// TIA Portal V19 export
FUNCTION_BLOCK "A0302_Manager_FB"   // FB51, LAD
// stored: MemoryReserve 100, SetENOAutomatically false
   VAR_INPUT
      AreaInterface : "AreaInterface";
      DataIn : Struct
         SemiAut_Pb : Bool;
      END_STRUCT;
      CIn : Struct
         P5 : Struct
            Sollevatori { ExternalAccessible := 'False'; ExternalVisible := 'False'; ExternalWritable := 'False'} : "ValveMachine_COut";
            Spintore_Lat : Struct
               Spin_Lat1 : Struct
                  Standstill : Bool;
                  Rest_CheckNext : Bool;
                  Work_CheckNext : Bool;
                  Rest : Bool;
                  Work : Bool;
               END_STRUCT;
               Spin_Lat2 : Struct
                  Standstill : Bool;
                  Rest_CheckNext : Bool;
                  Work_CheckNext : Bool;
                  Rest : Bool;
                  Work : Bool;
               END_STRUCT;
            END_STRUCT;
            SpintoreLong { ExternalAccessible := 'False'; ExternalVisible := 'False'; ExternalWritable := 'False'} : Struct   // Spintore Longitudinale
               Ax : "Positioning_EPOS_Machine_COut";
               Ax_Sts : Struct
                  PosAttesa_Reached : Bool;
                  PosFineSpinta_Reached : Bool;
               END_STRUCT;
               Spintore : "ValveMachine_COut";
               Vrt : "ValveMachine_COut";
               Orz : "ValveMachine_COut";
               Sens : Struct
                  FTC_FuoriIngombro : Bool;
               END_STRUCT;
            END_STRUCT;
         END_STRUCT;
         Bordatrice : Struct
            Ax : "Positioning_EPOS_Machine_COut";
            Sts : Struct
               PosTargetEnable : Bool;
               PosTarget_Reached : Bool;
               In_W_Pos : Bool;
               AtRest : Bool;
            END_STRUCT;
            Sens : Struct
               FTC_Ingresso : Bool;   // 1833SQ1 - I46.0 (Predisposta - usiamo la 1614BF1)
               FTC_Uscita : Bool;
            END_STRUCT;
         END_STRUCT;
         Rulliera { ExternalAccessible := 'False'; ExternalVisible := 'False'; ExternalWritable := 'False'} : Struct
            Ax_1 : "SpeedMachine_COut";
            Ax_2 : "SpeedMachine_COut";
            Centraggio : "ValveMachine_COut";   // Chiusura Centratori
            Sollevamento : "ValveMachine_COut";   // Solleva centratori
            Coda : Struct
               Sens : Struct
                  FTC_Rall : Bool;   // Sensori presenza materiale banco rallentamento ingresso
                  FTC_Prox_Ing : Bool;   // Sensori presenza materiale banco limite ingresso
               END_STRUCT;
            END_STRUCT;
            Centro : Struct
               Sens : Struct
                  FTC_Centrale : Bool;
               END_STRUCT;
            END_STRUCT;
         END_STRUCT;
         CarroPareggCoda { ExternalAccessible := 'False'; ExternalVisible := 'False'; ExternalWritable := 'False'} : Struct
            Ax_InWPos : Bool;
            Ax : "Positioning_DOL_Machine_COut";
            Bloccaggio : "ValveMachine_COut";
            BattutaVerticale : "ValveMachine_COut";
            PareggiatoreLong : "ValveMachine_COut";
            Sens : Struct
               FTC_Ingombro_Ing : Bool;   // FTC fuori ingombro lato ingresso al carro pareggiatore di coda
               FTC_Ingombro_Out : Bool;   // FTC fuori ingombro lato uscita al carro pareggiatore di coda
               PresenzaMat : Bool;   // FC presenza materiale agganciato
               PosPareggLong : Struct
                  Value : LReal;
                  CheckMeasure : Bool;
                  Standstill : Bool;
               END_STRUCT;
            END_STRUCT;
         END_STRUCT;
         CarroPareggTesta { ExternalAccessible := 'False'; ExternalVisible := 'False'; ExternalWritable := 'False'} : Struct
            Ax_InWPos : Bool;
            Ax : "Positioning_DOL_Machine_COut";
            Bloccaggio : "ValveMachine_COut";
            Centraggio : "ValveMachine_COut";
            Sollevatore : "ValveMachine_COut";
            Sens : Struct
               FTC_Ingombro_Ing : Bool;   // FTC fuori ingombro lato ingresso al carro pareggiatore di testa - Rallentamento rulliera
               FTC_Prox_Ls : Bool;   // FTC sensore presenza materiale banco limite ingresso
               PresenzaMat : Bool;   // FC presenza materiale agganciato
            END_STRUCT;
         END_STRUCT;
         Manipolatori : Struct
            Testa : Struct
               Ax : "Positioning_EPOS_Machine_COut";
               Sollevatore : "ValveMachine_COut";
               Magnete : "ValveMachine_COut";
            END_STRUCT;
            Coda : Struct
               Ax : "Positioning_EPOS_Machine_COut";
               Sollevatore : "ValveMachine_COut";
               Magnete : "ValveMachine_COut";
            END_STRUCT;
            InPos_Prelievo : Bool;
            InPos_BancoScarto : Bool;
            InPos_BancoA0303 : Bool;
         END_STRUCT;
         Spalle : Struct
            Coda : Struct
               Ax : "Positioning_DOL_Machine_COut";
            END_STRUCT;
            Testa : Struct
               Ax : "Positioning_DOL_Machine_COut";
            END_STRUCT;
         END_STRUCT;
         Banco_A0303 : Struct
            ReadyToRecive : Bool;   // Consenso da Stazione A0303 a ricevere il pezzo buono misurato
         END_STRUCT;
         ProdManager : "Prod_Beam_Ctrl";
      END_STRUCT;
   END_VAR
   VAR_OUTPUT
      MachineInterface : "MachineInterface";
      COut : Struct
         HU : Struct
            EnableStopDoorOpeningReq : Bool;
            EnableStopInPhase : Bool;
            EnableStopProgrammed : Bool;
            Control_ON : Bool;
            Rest : Bool;
            Work : Bool;
         END_STRUCT;
         SpintoreLong : Struct
            EnableStopDoorOpeningReq : Bool;
            EnableStopInPhase : Bool;
            EnableStopProgrammed : Bool;
            Control_ON : Bool;
            REST_Req : Bool;
            WORK_Req : Bool;
            Rest : Bool;
            Work : Bool;
         END_STRUCT;
         Bordatrice : Struct
            Ax : "Positioning_EPOS_Machine_Manager";
            Sts : Struct
               PosTarget_Reached : Bool;
               AtRest : Bool;
            END_STRUCT;
            DataOut : "Positioning_EPOS_Machine_DataOut";
            Rest_Req : Bool;
            Work_Req : Bool;
         END_STRUCT;
         Rulliera : Struct
            Ax_1 : "SpeedMachine_CIn_Manager";
            Ax_2 : "SpeedMachine_CIn_Manager";
            Centratori : Struct   // Chiusura Centratori
               Sollevamento : "ValveMachine_Manager";
               Centraggio : "ValveMachine_Manager";
            END_STRUCT;
            Ax_1_Frw_Req : Bool;
            Ax_1_Brw_Req : Bool;
            Ax_2_Frw_Req : Bool;
            Ax_2_Brw_Req : Bool;
         END_STRUCT;
         CarroPareggCoda : Struct
            EnableStopDoorOpeningReq : Bool;
            EnableStopInPhase : Bool;
            EnableStopProgrammed : Bool;
            Control_ON : Bool;
            MoveToPos : Bool;
            Pos : LReal;
            Speed : LReal;
            Bloccaggio : Struct
               Rest : Bool;
               Work : Bool;
            END_STRUCT;
            BattutaVrt : Struct
               Rest : Bool;
               Work : Bool;
            END_STRUCT;
            PareggLong : Struct
               Rest : Bool;
               Work : Bool;
            END_STRUCT;
         END_STRUCT;
         CarroPareggTesta : Struct
            EnableStopDoorOpeningReq : Bool;
            EnableStopInPhase : Bool;
            EnableStopProgrammed : Bool;
            Control_ON : Bool;
            MoveToPos : Bool;
            Pos : LReal;
            Speed : LReal;
            Bloccaggio : "OP_PB";
            Sollevamento : "OP_PB";
            Centraggio : "OP_PB";
         END_STRUCT;
         Manipolatori : Struct
            Ax : Struct
               EnableStopDoorOpeningReq : Bool;
               EnableStopInPhase : Bool;
               EnableStopProgrammed : Bool;
               Control_ON : Bool;
               MoveToPos : Bool;
               Pos : LReal;
               Vel : LReal;
               Acc : LReal;
               Dec : LReal;
            END_STRUCT;
            Sollevatori : "OP_PB";
            Magneti : "OP_PB";
         END_STRUCT;
      END_STRUCT;
   END_VAR
   VAR_IN_OUT
      Par : Struct
         CarroPareggCoda : Struct
            Delay_StartMove : Time;
            Preset : LReal;
         END_STRUCT;
         CarroPareggTesta : Struct
            Delay_StartMove : Time;
            Preset : LReal;
         END_STRUCT;
         Cremaliera : Struct
            Modulo : LReal;
            Passo : LReal;
         END_STRUCT;
      END_STRUCT;
   END_VAR
   VAR
      Alarm : Struct
         Qlty_Unknow : Bool;   // Allarme pezzo sconosciuto
         ToCheckList_Full : Bool;
         WrongReadPz_ManipBasso : Bool;
         Pz_NonPareggiabile : Bool;
         STOP_FineTurno : Bool;
         STOP_End_Of_Proroduction : Bool;
         STOP_ControlloQualita : Bool;
      END_STRUCT;
      Warning : Struct
         CheckBancoAccumulo : Bool;
      END_STRUCT;
      Sts : Struct
         SemiAut : Struct
            ON : Bool;
            Request : Bool;
            MaterialFrw : Bool;
         END_STRUCT;
         CarroPareggTesta : Struct
            InCyclePos : Bool;
         END_STRUCT;
         CarroPareggCoda : Struct
            InCyclePos : Bool;
         END_STRUCT;
         Attrezzamento : Struct
            Ready : Bool;
            FindNewID : Bool;
            RequestNewPosition : Bool;
            OLD_OID : DInt;
         END_STRUCT;
         BTrk : Struct
            A0302Exit_Actual_O_ID : DInt;
            BLen_Paregg : Real;
            Last_Misure1Paregg : Real;
            Last_Misure2Paregg : Real;
            A0302Entry_Absence : Bool;
            A0302Exit_Absence : Bool;
            ZoneA0302Entry_Empty : Bool;
            ZoneA0302Exit_Empty : Bool;
            A0302_CheckBancoAccumulo : Bool;
            Waiting_A0302_Recive : Bool;
         END_STRUCT;
         AlarmsPresence : Bool;
         WarningsPresence : Bool;
         IsStandstill : Bool;
      END_STRUCT;
      Ctrl : Struct
         Stop : Bool;
         TRK : Struct
            BTrk : Struct
               "P5.1_To_LongPosAttesa" : Bool;
               "P5.2_LongPosAttesa_TO_Spintore" : Bool;
               "P5.2_Spintore_TO_ExitA031" : Bool;
               "P5.2_ExitA031_To_IngBord" : Bool;
               "P5.2_Ax_MoveToPosAttesa" : Bool;
               "P5.2_Ax_PreparingPosAttesa" : Bool;
               "P5.2_Ax_MoveToPosSpinta" : Bool;
               SpinBord_In_To_Bord_In : Bool;
               Bordatrice_In_To_Out : Bool;   // il pezzo ha raggiunto il sensore di uscita della bordatrice (xxxSQx) (salvataggio posizione asse bordatrice)
               Bordatrice_Out_To_PareggCodaUp : Bool;   // Il pezzo è in uscita della bordatrice e la posizione target non è limitata perchè il pareggiamento di coda è alto
               Bordatrice_Out_To_PareggCodaDown : Bool;   // Il pezzo è in uscita della bordatrice ma la posizione target è limitata per non collidere con il pareggiamento di coda basso
               Rulliera_Start_Brw : Bool;
               Rulliera_Ax_1_Start_Frw : Bool;
               Rulliera_Ax_2_Start_Frw : Bool;
               RulliereVode : Bool;
               PCodaDown_TO_Rulli_PCodaDown : Bool;   // Pezzo su rulliera (1) + pareggiatore coda basso quindi quando incontra sensore (1,2) deve rallentare
               PCodaDown_TO_RALL_Rulli_PCodaDown : Bool;   // Pezzo su rulliera (1) + pareggiatore coda basso e ha incontrato sensore (1,2) di rallentamento
               PCodaDown_TO_STOP_PCodaDown : Bool;   // Pezzo su rulliera (1) + pareggiatore coda basso e ha incontrato sensore (3) di stop
               STOP_PCodaDown_TO_PCoda_Up : Bool;   // Pezzo su rulliera (1) + pareggiatore coda alto quindi può muoversi liberamente
               "PareggCodaUp_To_Rull-PrimaPareggCodaAltro" : Bool;
               PCoda_Up_TO_PCoda_UP_S3 : Bool;   // Pezzo su rulliera (1) + pareggiatore coda alto ed ha incontrato il sensore 3 (in ingresso al pareg.)
               PCoda_UP_S3_TO_PCoda_UP_S4 : Bool;   // Pezzo su rulliera (1) + pareggiatore coda alto ed ha incontrato il sensore 4 (in uscita al pareg.)
               PCoda_UP_S4_TO_PCoda_DownCnd : Bool;   // Pezzo su rulliera (1/2) + pareggiatore coda che è alto ed ha liberato il sensore 4-> Pareg. può andare basso (posizione di lavoro)
               PCoda_Beam_TO_PTesta : Bool;   // Pezzo su rulliera (1/2) tra il pareggiatore di testa e quello di coda
               Beam_TO_Stop_PTesta : Bool;   // Pezzo su rulliera (1/2) + ha incontrato il sensore 5 su pareggiatore di testa
               "Stop_PTesta_TO_Rull-Centratori" : Bool;   // Pezzo su rulliera (1/2) tra i pareggiatori + centratori a lavoro
               "Rull-Centratori_TO_Cnd_PareggCoda" : Bool;   // Pezzo su rulliera (1/2) tra i pareggiatori (quello di coda è basso) + centratori a lavoro
               Cnd_PareggCoda_TO_Pareggiato : Bool;   // Pezzo su rulliera (1/2) tra i pareggiatori e paregiatura di coda eseguito lavoro cilindro idraulico (ora si sa la misura del pezzo, si può mettere utenze in attesa del prossimo pezzo)
               Check_Tolleranza_BLen_Qlty : Bool;
               Pareggiato_TO_PresaBasso : Bool;   // Pezzo su magneti del manipolatore basso in posizione di presa.
               PresaBasso_TO_PresaAlto : Bool;   // Pezzo su magneti del manipolatore alto in posizione di presa.
               PresaAlto_To_CheckOut_BadQlty : Bool;   // Pezzo su magneti del manipolatore alto in posizione di uscita perchè non conforme
               CheckOut_BadQlty_UP_MoveToPos : Bool;   // Ho il pezzo in presa alta > vado in posizione uscita banco scarto
               PresaAlto_To_CheckOut_GoodQlty : Bool;   // Pezzo su magneti del manipolatore alto in posizione per deposito su A0303
               CheckOut_GoodQlty_UP_MoveToPos : Bool;   // Ho il pezzo in presa alta > vado in posizione uscita banco A0303
               CheckOut_BadQlty_UP_To_DOWN : Bool;   // Pezzo su magneti del manipolatore basso in posizione di uscita perchè non conforme
               CheckOut_BadQlty_DOWN_To_Sgancia : Bool;
               CheckOut_GoodQlty_UP_To_DOWN : Bool;   // Pezzo su magneti del manipolatore basso in posizione per deposito su A0303
               CheckOut_GoodQlty_DOWN_To_Sgancia : Bool;
               Manipolatori_Return_ToPrelievo : Bool;   // Ritorno degli assi manipolatore a zero e / o a prelievo
            END_STRUCT;
            BTrk_ToCheck : Struct
               ClearList : Bool;
               QtyClear_RetVal : Bool;
               Prelievo_RecondGood : Bool;   // Attivo durante la fase di posizionamento manuale del Beam fino a quando il manipolatore lo prende
               RecG_InPos_Centraggio : Bool;   // Beam ricondizionato posizionato su rulliera da centrare
               RegG_InPos_ReadyPickUp : Bool;
            END_STRUCT;
         END_STRUCT;
         SpintoreLong : Struct
            Rest : Bool;
            Work : Bool;
            MoveAttesaDisable : Bool;
         END_STRUCT;
         Bordatrice : Struct
            Run : Bool;
         END_STRUCT;
         Rulliera : Struct
            Ax_1_Vel_Bord : Bool;
            Ax_2_Vel_Bord : Bool;
            Ax_1_Lenta_CarroCoda : Bool;
            Ax_1_2_Vel_CarroTesta : Bool;
            Ax_1_2_Vel_ZeroTesta : Bool;
            Ax_1_2_Vel_Appoggio : Bool;
            Ax_1_2_End_VelZero : Bool;
            Ax_2_MemoRall : Bool;
            SP_TimeMemoRall : Time;
            TON_RitardoRallenta : IEC_TIMER;
            Centraggio : Struct
               Rest : Bool;
               Work : Bool;
            END_STRUCT;
            Sollevamento : Struct
               Rest : Bool;
               Work : Bool;
            END_STRUCT;
         END_STRUCT;
         CarroPareggCoda : Struct
            Ax : Struct
               MoveToPos : Bool;
               Pos : LReal;
            END_STRUCT;
            Bloccaggio : Struct
               Rest : Bool;
               Work : Bool;
            END_STRUCT;
            BattutaVerticale : Struct
               Rest : Bool;
               Work : Bool;
            END_STRUCT;
            PareggiatoreLong : Struct
               Rest : Bool;
               Work : Bool;
            END_STRUCT;
            MisuraPzPareggiato : Bool;
         END_STRUCT;
         CarroPareggTesta : Struct
            Ax : Struct
               MoveToPos : Bool;
               Pos : LReal;
            END_STRUCT;
            Bloccaggio : Struct
               Rest : Bool;
               Work : Bool;
            END_STRUCT;
            Sollevatore : Struct
               Rest : Bool;
               Work : Bool;
            END_STRUCT;
            Centraggio : Struct
               Rest : Bool;
               Work : Bool;
            END_STRUCT;
         END_STRUCT;
         Manipolatori : Struct
            Ax : Struct
               MoveToPos : Bool;
               Pos : LReal;
            END_STRUCT;
            Sollevatori : Struct
               Rest : Bool;
               Work : Bool;
            END_STRUCT;
            Magneti : Struct
               Rest : Bool;
               Work : Bool;
            END_STRUCT;
         END_STRUCT;
      END_STRUCT;
      HMI : Struct
         PlsClear_ListToCheck : Bool;
      END_STRUCT;
      BTrk_A0302_Exit_Item : Struct
         BLean : Real;
         W_A : Real;
         Tol_Max : Real;
         Tol_Min : Real;
         Good { ExternalAccessible := 'False'; ExternalVisible := 'False'; ExternalWritable := 'False'} : Bool;
         ToCheckLen { ExternalAccessible := 'False'; ExternalVisible := 'False'; ExternalWritable := 'False'} : Bool;
      END_STRUCT;
      BTrk_ListToCheck : Struct
         Recond : Struct
            Found : Bool;
            Nr_B : Int;
         END_STRUCT;
      END_STRUCT;
      OffsetCarri : Struct
         DaSpallaTesta : LReal;
         DaSpallaCoda : LReal;
      END_STRUCT;
      CarroTesta : Struct
         RimanenzaPos : LReal;
         PassoReq : LReal;
         PosBattutePz : LReal;
         SemiBeamLen : LReal;
         NrPassiReq : LReal;
      END_STRUCT;
      CarroCoda : Struct
         RimanenzaPos : LReal;
         PassoReq : LReal;
         PosBattutePz : LReal;
         SemiBeamLen : LReal;
         NrPassiReq : LReal;
      END_STRUCT;
      TON_AlarmWrongReadPz_Manip : IEC_TIMER;
      TON_Alarm_FTC_CarroCodaOut { S7_SetPoint := 'True'} : IEC_TIMER;
      TON_Stop { S7_SetPoint := 'True'} : IEC_TIMER;
   END_VAR
   VAR_TEMP
      AUX : Struct
         SemiAut_Pb : Bool;
      END_STRUCT;
      i : Int;
      BTrk_A0302_EXIT_GetData : Struct   // Appoggio struttura per lettura dati dal Mes
         indx : Int;   // Se trovato tra i TODO / ENDING / OUT questo è l'indice dove sono stati prelevati i dati
         Sts : Int;   // 0 = Non Trovato; 0 = ACT; 1 = TODO; 2=ENDING; 3 = OUT
         Item : "Prod_Item_small";
      END_STRUCT;
      DisableA0302 : Bool;
      PieceToCheck_Presence : Bool;
      CarroTestaCentraggio_Disable : Bool;
   END_VAR
   VAR CONSTANT
      OffsetGioco : Real := 2.0;   // Offset gioco carri durante lettura Pareggiamento pezzo
   END_VAR
   VAR_TEMP   // added for the SCL form of the ladder/FBD networks
      _w1 : Bool;
      _w2 : Bool;
      _w3 : Bool;
      _w4 : Bool;
      _w5 : Bool;
      _w6 : Bool;
      _w7 : Bool;
      _w8 : Bool;
      _w9 : Bool;
      _w10 : Bool;
      _w11 : Bool;
      _w12 : Bool;
      _w13 : Bool;
      _w14 : Bool;
      _w15 : Bool;
      _w16 : Bool;
      _w17 : Bool;
      _w18 : Bool;
      _w19 : Bool;
      _w20 : Bool;
   END_VAR
BEGIN

REGION Network 1 (SCL): = Area - Rst =
   IF #AreaInterface.RstAlarms THEN
       #Alarm.Qlty_Unknow := FALSE;
       #Alarm.ToCheckList_Full := FALSE;
       #Alarm.STOP_ControlloQualita := FALSE;
       #Alarm.STOP_FineTurno := FALSE;
       #Alarm.STOP_End_Of_Proroduction := FALSE;
   END_IF;

   IF #AreaInterface.RstAlarms AND #CIn.CarroPareggCoda.Sens.PresenzaMat AND #CIn.CarroPareggTesta.Sens.PresenzaMat
       AND #CIn.Manipolatori.Testa.Magnete.Work AND #CIn.Manipolatori.Coda.Magnete.Work THEN
       #Alarm.WrongReadPz_ManipBasso := FALSE;
   END_IF;

   IF #AreaInterface.RstAlarms AND NOT #CIn.CarroPareggCoda.Sens.FTC_Ingombro_Out THEN
       #Alarm.Pz_NonPareggiabile := FALSE;
   END_IF;
END_REGION

REGION Network 2: ******** CLEAR TRACKING ARRIVATO ********
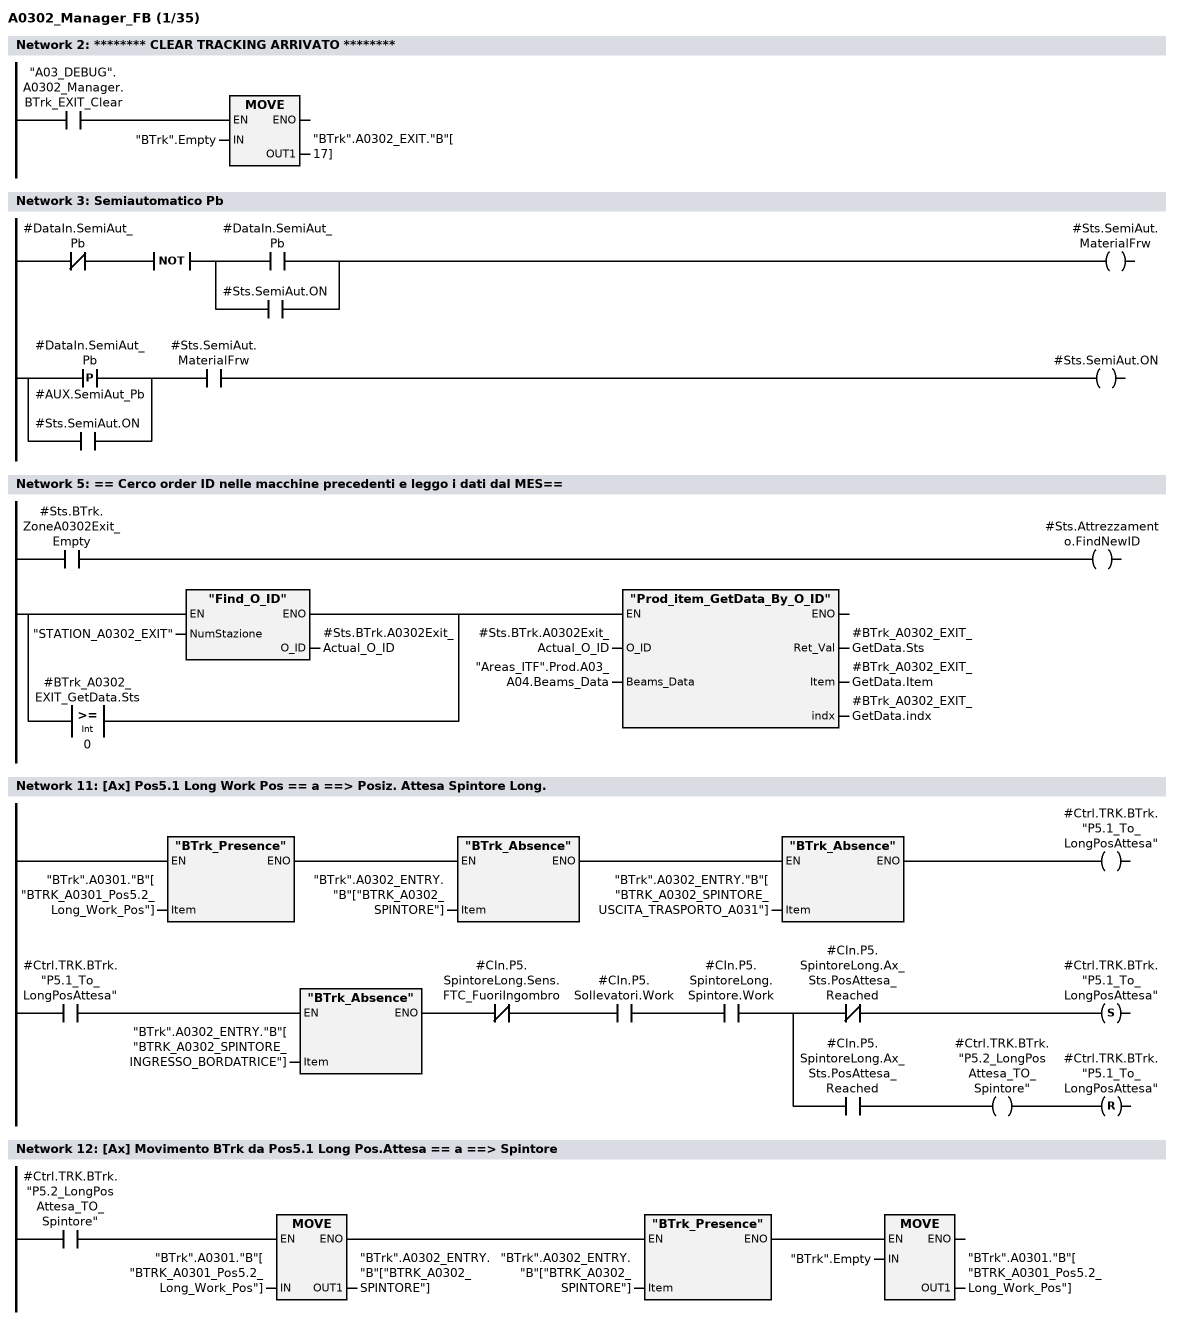
   RUNG wire#powerrail
      Contact( "A03_DEBUG".A0302_Manager.BTrk_EXIT_Clear )
      Move(in := "BTrk".Empty, out1 => "BTrk".A0302_EXIT."B"[17])
   END_RUNG
   // the same network as SCL:
   IF "A03_DEBUG".A0302_Manager.BTrk_EXIT_Clear THEN "BTrk".A0302_EXIT."B"[17] := "BTrk".Empty; END_IF;
END_REGION

REGION Network 3: Semiautomatico Pb
   RUNG wire#powerrail
      I_Contact( #DataIn.SemiAut_Pb )
      Not()
      wire#w1
      Contact( #DataIn.SemiAut_Pb )
      wire#w2
      Coil( #Sts.SemiAut.MaterialFrw )
   END_RUNG
   RUNG wire#w1
      Contact( #Sts.SemiAut.ON )
   END_RUNG wire#w2
   RUNG wire#powerrail
      P_Contact(operand := #DataIn.SemiAut_Pb, bit := #AUX.SemiAut_Pb)
      wire#w3
      Contact( #Sts.SemiAut.MaterialFrw )
      Coil( #Sts.SemiAut.ON )
   END_RUNG
   RUNG wire#powerrail
      Contact( #Sts.SemiAut.ON )
   END_RUNG wire#w3
   // the same network as SCL:
   #Sts.SemiAut.MaterialFrw := NOT (NOT #DataIn.SemiAut_Pb) AND (#DataIn.SemiAut_Pb OR #Sts.SemiAut.ON);
   #_w1 := #DataIn.SemiAut_Pb AND NOT #AUX.SemiAut_Pb;   // rising edge of #DataIn.SemiAut_Pb
   #AUX.SemiAut_Pb := #DataIn.SemiAut_Pb;
   #Sts.SemiAut.ON := (#_w1 OR #Sts.SemiAut.ON) AND #Sts.SemiAut.MaterialFrw;
END_REGION

REGION Network 5: == Cerco order ID nelle macchine precedenti e leggo i dati dal MES==
   RUNG wire#powerrail
      Contact( #Sts.BTrk.ZoneA0302Exit_Empty )
      Coil( #Sts.Attrezzamento.FindNewID )
   END_RUNG
   RUNG wire#powerrail
      "Find_O_ID"(NumStazione := "STATION_A0302_EXIT", O_ID => #Sts.BTrk.A0302Exit_Actual_O_ID)
      wire#w1
      "Prod_item_GetData_By_O_ID"(O_ID := #Sts.BTrk.A0302Exit_Actual_O_ID, Beams_Data := "Areas_ITF".Prod.A03_A04.Beams_Data, Ret_Val => #BTrk_A0302_EXIT_GetData.Sts, Item => #BTrk_A0302_EXIT_GetData.Item, indx => #BTrk_A0302_EXIT_GetData.indx)
   END_RUNG
   RUNG wire#powerrail
      { S7_Templates := "SrcType := Int" } GE_Contact(in1 := #BTrk_A0302_EXIT_GetData.Sts, in2 := 0)
   END_RUNG wire#w1
   // the same network as SCL:
   #Sts.Attrezzamento.FindNewID := #Sts.BTrk.ZoneA0302Exit_Empty;
   "Find_O_ID"(NumStazione := "STATION_A0302_EXIT", O_ID => #Sts.BTrk.A0302Exit_Actual_O_ID, ENO => #_w1);
   IF #_w1 OR (#BTrk_A0302_EXIT_GetData.Sts >= 0) THEN
       #BTrk_A0302_EXIT_GetData.Sts := "Prod_item_GetData_By_O_ID"(O_ID := #Sts.BTrk.A0302Exit_Actual_O_ID,
                               Beams_Data := "Areas_ITF".Prod.A03_A04.Beams_Data,
                               Item => #BTrk_A0302_EXIT_GetData.Item,
                               indx => #BTrk_A0302_EXIT_GetData.indx);
   END_IF;
END_REGION

REGION Network 6 (SCL): == Richiesta nuovo posizionamento carri Testa/Coda per cambio Traking ==

   //Se ho O_ID <> e non sono vuoto attivo avviso di attesa zona A0302 vuota
   IF (#Sts.BTrk.A0302Exit_Actual_O_ID <> #Sts.Attrezzamento.OLD_OID) OR (NOT #Sts.BTrk.ZoneA0302Exit_Empty OR NOT #Sts.BTrk.ZoneA0302Entry_Empty)THEN
       #Sts.BTrk.Waiting_A0302_Recive := TRUE;

   ELSIF (#Sts.BTrk.A0302Exit_Actual_O_ID = #Sts.Attrezzamento.OLD_OID) OR ( #Sts.BTrk.ZoneA0302Exit_Empty AND #Sts.BTrk.ZoneA0302Entry_Empty) THEN
       #Sts.BTrk.Waiting_A0302_Recive := FALSE;

   END_IF;

   //Se ho O_ID <> e sono vuoto aggiorno vecchio O_ID 
   IF (#Sts.BTrk.A0302Exit_Actual_O_ID <> #Sts.Attrezzamento.OLD_OID) AND #Sts.BTrk.ZoneA0302Exit_Empty AND #Sts.BTrk.ZoneA0302Entry_Empty THEN
       #Sts.Attrezzamento.OLD_OID := #Sts.BTrk.A0302Exit_Actual_O_ID;
   END_IF;
END_REGION

REGION Network 7 (SCL): == Compilo i dati del btrk in base all'order ID in arrivo ==

   IF #BTrk_A0302_EXIT_GetData.Sts >= 0 THEN

       "BTrk".A0302_EXIT.O_ID:="BTrk".A0302_ENTRY.O_ID := #Sts.Attrezzamento.OLD_OID;
       "BTrk".A0302_EXIT.Beam_Len := "BTrk".A0302_ENTRY.Beam_Len := #BTrk_A0302_EXIT_GetData.Item.Beams_Len;
       "BTrk".A0302_EXIT.Beam_W_A := "BTrk".A0302_ENTRY.Beam_W_A := #BTrk_A0302_EXIT_GetData.Item.Beams_W_A;
       "BTrk".A0302_EXIT.Beam_H_B := "BTrk".A0302_ENTRY.Beam_H_B := #BTrk_A0302_EXIT_GetData.Item.Beams_H_B;

   ELSE
           "BTrk".A0302_EXIT.O_ID := "BTrk".A0302_ENTRY.O_ID := "BTrk".A0301.O_ID := -1;
           "BTrk".A0302_EXIT.Beam_Len := "BTrk".A0302_ENTRY.Beam_Len := -1.0;
           "BTrk".A0302_EXIT.Beam_W_A := "BTrk".A0302_ENTRY.Beam_W_A := -1.0;
           "BTrk".A0302_EXIT.Beam_H_B := "BTrk".A0302_ENTRY.Beam_H_B := -1.0;
   END_IF;
END_REGION

REGION Network 8 (SCL): == Richiesta nuovo posizionamento x cambio Order ID ==

   #Sts.Attrezzamento.RequestNewPosition := ("BTrk".A0302_EXIT.O_ID <> -1)
   AND (#BTrk_A0302_EXIT_GetData.Sts >= 0)
   AND (#BTrk_A0302_EXIT_GetData.Item.Beam_Code = 1)
   AND #Sts.Attrezzamento.FindNewID
   AND NOT #Sts.Attrezzamento.Ready
   AND NOT #BTrk_ListToCheck.Recond.Found
   AND (NOT #CIn.CarroPareggCoda.Ax_InWPos OR NOT #CIn.CarroPareggTesta.Ax_InWPos);
END_REGION

REGION Network 10: <<<< SPINTORE LONGITUDINALE >>>>
END_REGION

REGION Network 11: [Ax] Pos5.1 Long Work Pos == a ==> Posiz. Attesa Spintore Long.
   RUNG wire#powerrail
      "BTrk_Presence"(Item := "BTrk".A0301."B"["BTRK_A0301_Pos5.2_Long_Work_Pos"])
      "BTrk_Absence"(Item := "BTrk".A0302_ENTRY."B"["BTRK_A0302_SPINTORE"])
      "BTrk_Absence"(Item := "BTrk".A0302_ENTRY."B"["BTRK_A0302_SPINTORE_USCITA_TRASPORTO_A031"])
      Coil( #Ctrl.TRK.BTrk."P5.1_To_LongPosAttesa" )
   END_RUNG
   RUNG wire#powerrail
      Contact( #Ctrl.TRK.BTrk."P5.1_To_LongPosAttesa" )
      "BTrk_Absence"(Item := "BTrk".A0302_ENTRY."B"["BTRK_A0302_SPINTORE_INGRESSO_BORDATRICE"])
      I_Contact( #CIn.P5.SpintoreLong.Sens.FTC_FuoriIngombro )
      Contact( #CIn.P5.Sollevatori.Work )
      Contact( #CIn.P5.SpintoreLong.Spintore.Work )
      wire#w1
      I_Contact( #CIn.P5.SpintoreLong.Ax_Sts.PosAttesa_Reached )
      S_Coil( #Ctrl.TRK.BTrk."P5.1_To_LongPosAttesa" )
   END_RUNG
   RUNG wire#w1
      Contact( #CIn.P5.SpintoreLong.Ax_Sts.PosAttesa_Reached )
      Coil( #Ctrl.TRK.BTrk."P5.2_LongPosAttesa_TO_Spintore" )
      R_Coil( #Ctrl.TRK.BTrk."P5.1_To_LongPosAttesa" )
   END_RUNG
   // the same network as SCL:
   "BTrk_Presence"(Item := "BTrk".A0301."B"["BTRK_A0301_Pos5.2_Long_Work_Pos"], ENO => #_w1);
   "BTrk_Absence"(EN := #_w1, Item := "BTrk".A0302_ENTRY."B"["BTRK_A0302_SPINTORE"], ENO => #_w2);
   "BTrk_Absence"(EN := #_w2,
                  Item := "BTrk".A0302_ENTRY."B"["BTRK_A0302_SPINTORE_USCITA_TRASPORTO_A031"],
                  ENO => #_w3);
   #Ctrl.TRK.BTrk."P5.1_To_LongPosAttesa" := #_w3;
   "BTrk_Absence"(EN := #Ctrl.TRK.BTrk."P5.1_To_LongPosAttesa",
                  Item := "BTrk".A0302_ENTRY."B"["BTRK_A0302_SPINTORE_INGRESSO_BORDATRICE"],
                  ENO => #_w4);
   #_w5 := #_w4 AND NOT #CIn.P5.SpintoreLong.Sens.FTC_FuoriIngombro AND #CIn.P5.Sollevatori.Work AND #CIn.P5.SpintoreLong.Spintore.Work;
   IF #_w5 AND NOT #CIn.P5.SpintoreLong.Ax_Sts.PosAttesa_Reached THEN
       #Ctrl.TRK.BTrk."P5.1_To_LongPosAttesa" := TRUE;
   END_IF;
   #Ctrl.TRK.BTrk."P5.2_LongPosAttesa_TO_Spintore" := #_w5 AND #CIn.P5.SpintoreLong.Ax_Sts.PosAttesa_Reached;
   IF #Ctrl.TRK.BTrk."P5.2_LongPosAttesa_TO_Spintore" THEN
       #Ctrl.TRK.BTrk."P5.1_To_LongPosAttesa" := FALSE;
   END_IF;
END_REGION

REGION Network 12: [Ax] Movimento BTrk da Pos5.1 Long Pos.Attesa == a ==> Spintore
   RUNG wire#powerrail
      Contact( #Ctrl.TRK.BTrk."P5.2_LongPosAttesa_TO_Spintore" )
      Move(in := "BTrk".A0301."B"["BTRK_A0301_Pos5.2_Long_Work_Pos"], out1 => "BTrk".A0302_ENTRY."B"["BTRK_A0302_SPINTORE"])
      "BTrk_Presence"(Item := "BTrk".A0302_ENTRY."B"["BTRK_A0302_SPINTORE"])
      Move(in := "BTrk".Empty, out1 => "BTrk".A0301."B"["BTRK_A0301_Pos5.2_Long_Work_Pos"])
   END_RUNG
   // the same network as SCL:
   IF #Ctrl.TRK.BTrk."P5.2_LongPosAttesa_TO_Spintore" THEN
       "BTrk".A0302_ENTRY."B"["BTRK_A0302_SPINTORE"] := "BTrk".A0301."B"["BTRK_A0301_Pos5.2_Long_Work_Pos"];
   END_IF;
   "BTrk_Presence"(EN := #Ctrl.TRK.BTrk."P5.2_LongPosAttesa_TO_Spintore",
                   Item := "BTrk".A0302_ENTRY."B"["BTRK_A0302_SPINTORE"],
                   ENO => #_w1);
   IF #_w1 THEN "BTrk".A0301."B"["BTRK_A0301_Pos5.2_Long_Work_Pos"] := "BTrk".Empty; END_IF;
END_REGION

REGION Network 13: [Ax] Movimento BTrk da A3202 Spintore ==a==> Uscita Trasporto A031
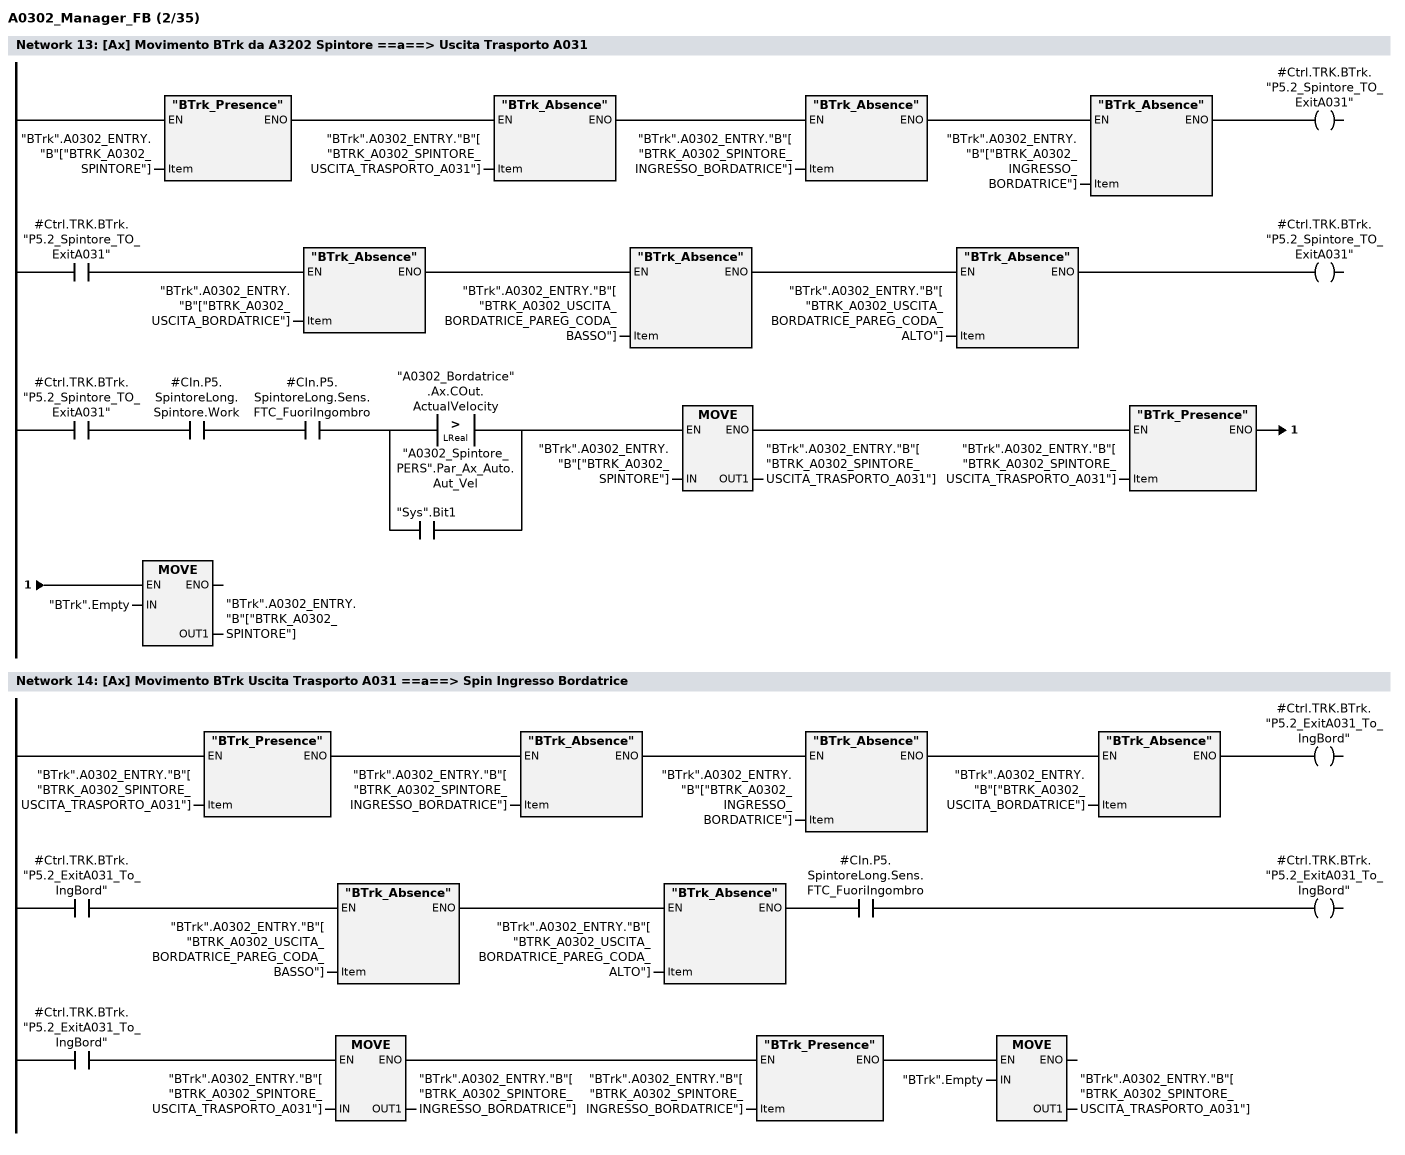
   RUNG wire#powerrail
      "BTrk_Presence"(Item := "BTrk".A0302_ENTRY."B"["BTRK_A0302_SPINTORE"])
      "BTrk_Absence"(Item := "BTrk".A0302_ENTRY."B"["BTRK_A0302_SPINTORE_USCITA_TRASPORTO_A031"])
      "BTrk_Absence"(Item := "BTrk".A0302_ENTRY."B"["BTRK_A0302_SPINTORE_INGRESSO_BORDATRICE"])
      "BTrk_Absence"(Item := "BTrk".A0302_ENTRY."B"["BTRK_A0302_INGRESSO_BORDATRICE"])
      Coil( #Ctrl.TRK.BTrk."P5.2_Spintore_TO_ExitA031" )
   END_RUNG
   RUNG wire#powerrail
      Contact( #Ctrl.TRK.BTrk."P5.2_Spintore_TO_ExitA031" )
      "BTrk_Absence"(Item := "BTrk".A0302_ENTRY."B"["BTRK_A0302_USCITA_BORDATRICE"])
      "BTrk_Absence"(Item := "BTrk".A0302_ENTRY."B"["BTRK_A0302_USCITA_BORDATRICE_PAREG_CODA_BASSO"])
      "BTrk_Absence"(Item := "BTrk".A0302_ENTRY."B"["BTRK_A0302_USCITA_BORDATRICE_PAREG_CODA_ALTO"])
      Coil( #Ctrl.TRK.BTrk."P5.2_Spintore_TO_ExitA031" )
   END_RUNG
   RUNG wire#powerrail
      Contact( #Ctrl.TRK.BTrk."P5.2_Spintore_TO_ExitA031" )
      Contact( #CIn.P5.SpintoreLong.Spintore.Work )
      Contact( #CIn.P5.SpintoreLong.Sens.FTC_FuoriIngombro )
      wire#w1
      { S7_Templates := "SrcType := LReal" } GT_Contact(in1 := "A0302_Bordatrice".Ax.COut.ActualVelocity, in2 := "A0302_Spintore_PERS".Par_Ax_Auto.Aut_Vel)
      wire#w2
      Move(in := "BTrk".A0302_ENTRY."B"["BTRK_A0302_SPINTORE"], out1 => "BTrk".A0302_ENTRY."B"["BTRK_A0302_SPINTORE_USCITA_TRASPORTO_A031"])
      "BTrk_Presence"(Item := "BTrk".A0302_ENTRY."B"["BTRK_A0302_SPINTORE_USCITA_TRASPORTO_A031"])
      Move(in := "BTrk".Empty, out1 => "BTrk".A0302_ENTRY."B"["BTRK_A0302_SPINTORE"])
   END_RUNG
   RUNG wire#w1
      Contact( "Sys".Bit1 )
   END_RUNG wire#w2
   // the same network as SCL:
   "BTrk_Presence"(Item := "BTrk".A0302_ENTRY."B"["BTRK_A0302_SPINTORE"], ENO => #_w1);
   "BTrk_Absence"(EN := #_w1,
                  Item := "BTrk".A0302_ENTRY."B"["BTRK_A0302_SPINTORE_USCITA_TRASPORTO_A031"],
                  ENO => #_w2);
   "BTrk_Absence"(EN := #_w2,
                  Item := "BTrk".A0302_ENTRY."B"["BTRK_A0302_SPINTORE_INGRESSO_BORDATRICE"],
                  ENO => #_w3);
   "BTrk_Absence"(EN := #_w3, Item := "BTrk".A0302_ENTRY."B"["BTRK_A0302_INGRESSO_BORDATRICE"], ENO => #_w4);
   #Ctrl.TRK.BTrk."P5.2_Spintore_TO_ExitA031" := #_w4;
   "BTrk_Absence"(EN := #Ctrl.TRK.BTrk."P5.2_Spintore_TO_ExitA031",
                  Item := "BTrk".A0302_ENTRY."B"["BTRK_A0302_USCITA_BORDATRICE"],
                  ENO => #_w5);
   "BTrk_Absence"(EN := #_w5,
                  Item := "BTrk".A0302_ENTRY."B"["BTRK_A0302_USCITA_BORDATRICE_PAREG_CODA_BASSO"],
                  ENO => #_w6);
   "BTrk_Absence"(EN := #_w6,
                  Item := "BTrk".A0302_ENTRY."B"["BTRK_A0302_USCITA_BORDATRICE_PAREG_CODA_ALTO"],
                  ENO => #_w7);
   #Ctrl.TRK.BTrk."P5.2_Spintore_TO_ExitA031" := #_w7;
   IF #Ctrl.TRK.BTrk."P5.2_Spintore_TO_ExitA031" AND #CIn.P5.SpintoreLong.Spintore.Work AND #CIn.P5.SpintoreLong.Sens.FTC_FuoriIngombro AND (("A0302_Bordatrice".Ax.COut.ActualVelocity > "A0302_Spintore_PERS".Par_Ax_Auto.Aut_Vel) OR "Sys".Bit1) THEN
       "BTrk".A0302_ENTRY."B"["BTRK_A0302_SPINTORE_USCITA_TRASPORTO_A031"] := "BTrk".A0302_ENTRY."B"["BTRK_A0302_SPINTORE"];
   END_IF;
   "BTrk_Presence"(EN := #Ctrl.TRK.BTrk."P5.2_Spintore_TO_ExitA031" AND #CIn.P5.SpintoreLong.Spintore.Work AND #CIn.P5.SpintoreLong.Sens.FTC_FuoriIngombro AND (("A0302_Bordatrice".Ax.COut.ActualVelocity > "A0302_Spintore_PERS".Par_Ax_Auto.Aut_Vel) OR "Sys".Bit1),
                   Item := "BTrk".A0302_ENTRY."B"["BTRK_A0302_SPINTORE_USCITA_TRASPORTO_A031"],
                   ENO => #_w8);
   IF #_w8 THEN "BTrk".A0302_ENTRY."B"["BTRK_A0302_SPINTORE"] := "BTrk".Empty; END_IF;
END_REGION

REGION Network 14: [Ax] Movimento BTrk Uscita Trasporto A031 ==a==> Spin Ingresso Bordatrice
   RUNG wire#powerrail
      "BTrk_Presence"(Item := "BTrk".A0302_ENTRY."B"["BTRK_A0302_SPINTORE_USCITA_TRASPORTO_A031"])
      "BTrk_Absence"(Item := "BTrk".A0302_ENTRY."B"["BTRK_A0302_SPINTORE_INGRESSO_BORDATRICE"])
      "BTrk_Absence"(Item := "BTrk".A0302_ENTRY."B"["BTRK_A0302_INGRESSO_BORDATRICE"])
      "BTrk_Absence"(Item := "BTrk".A0302_ENTRY."B"["BTRK_A0302_USCITA_BORDATRICE"])
      Coil( #Ctrl.TRK.BTrk."P5.2_ExitA031_To_IngBord" )
   END_RUNG
   RUNG wire#powerrail
      Contact( #Ctrl.TRK.BTrk."P5.2_ExitA031_To_IngBord" )
      "BTrk_Absence"(Item := "BTrk".A0302_ENTRY."B"["BTRK_A0302_USCITA_BORDATRICE_PAREG_CODA_BASSO"])
      "BTrk_Absence"(Item := "BTrk".A0302_ENTRY."B"["BTRK_A0302_USCITA_BORDATRICE_PAREG_CODA_ALTO"])
      Contact( #CIn.P5.SpintoreLong.Sens.FTC_FuoriIngombro )
      Coil( #Ctrl.TRK.BTrk."P5.2_ExitA031_To_IngBord" )
   END_RUNG
   RUNG wire#powerrail
      Contact( #Ctrl.TRK.BTrk."P5.2_ExitA031_To_IngBord" )
      Move(in := "BTrk".A0302_ENTRY."B"["BTRK_A0302_SPINTORE_USCITA_TRASPORTO_A031"], out1 => "BTrk".A0302_ENTRY."B"["BTRK_A0302_SPINTORE_INGRESSO_BORDATRICE"])
      "BTrk_Presence"(Item := "BTrk".A0302_ENTRY."B"["BTRK_A0302_SPINTORE_INGRESSO_BORDATRICE"])
      Move(in := "BTrk".Empty, out1 => "BTrk".A0302_ENTRY."B"["BTRK_A0302_SPINTORE_USCITA_TRASPORTO_A031"])
   END_RUNG
   // the same network as SCL:
   "BTrk_Presence"(Item := "BTrk".A0302_ENTRY."B"["BTRK_A0302_SPINTORE_USCITA_TRASPORTO_A031"], ENO => #_w1);
   "BTrk_Absence"(EN := #_w1,
                  Item := "BTrk".A0302_ENTRY."B"["BTRK_A0302_SPINTORE_INGRESSO_BORDATRICE"],
                  ENO => #_w2);
   "BTrk_Absence"(EN := #_w2, Item := "BTrk".A0302_ENTRY."B"["BTRK_A0302_INGRESSO_BORDATRICE"], ENO => #_w3);
   "BTrk_Absence"(EN := #_w3, Item := "BTrk".A0302_ENTRY."B"["BTRK_A0302_USCITA_BORDATRICE"], ENO => #_w4);
   #Ctrl.TRK.BTrk."P5.2_ExitA031_To_IngBord" := #_w4;
   "BTrk_Absence"(EN := #Ctrl.TRK.BTrk."P5.2_ExitA031_To_IngBord",
                  Item := "BTrk".A0302_ENTRY."B"["BTRK_A0302_USCITA_BORDATRICE_PAREG_CODA_BASSO"],
                  ENO => #_w5);
   "BTrk_Absence"(EN := #_w5,
                  Item := "BTrk".A0302_ENTRY."B"["BTRK_A0302_USCITA_BORDATRICE_PAREG_CODA_ALTO"],
                  ENO => #_w6);
   #Ctrl.TRK.BTrk."P5.2_ExitA031_To_IngBord" := #_w6 AND #CIn.P5.SpintoreLong.Sens.FTC_FuoriIngombro;
   IF #Ctrl.TRK.BTrk."P5.2_ExitA031_To_IngBord" THEN
       "BTrk".A0302_ENTRY."B"["BTRK_A0302_SPINTORE_INGRESSO_BORDATRICE"] := "BTrk".A0302_ENTRY."B"["BTRK_A0302_SPINTORE_USCITA_TRASPORTO_A031"];
   END_IF;
   "BTrk_Presence"(EN := #Ctrl.TRK.BTrk."P5.2_ExitA031_To_IngBord",
                   Item := "BTrk".A0302_ENTRY."B"["BTRK_A0302_SPINTORE_INGRESSO_BORDATRICE"],
                   ENO => #_w7);
   IF #_w7 THEN "BTrk".A0302_ENTRY."B"["BTRK_A0302_SPINTORE_USCITA_TRASPORTO_A031"] := "BTrk".Empty; END_IF;
END_REGION

REGION Network 16: <<< GESTIONE MOVIMENTO SPINTORE LONGITUDINALE >>
END_REGION

REGION Network 17: [Ax] Spintore - Control - Pos. Fine Spinta
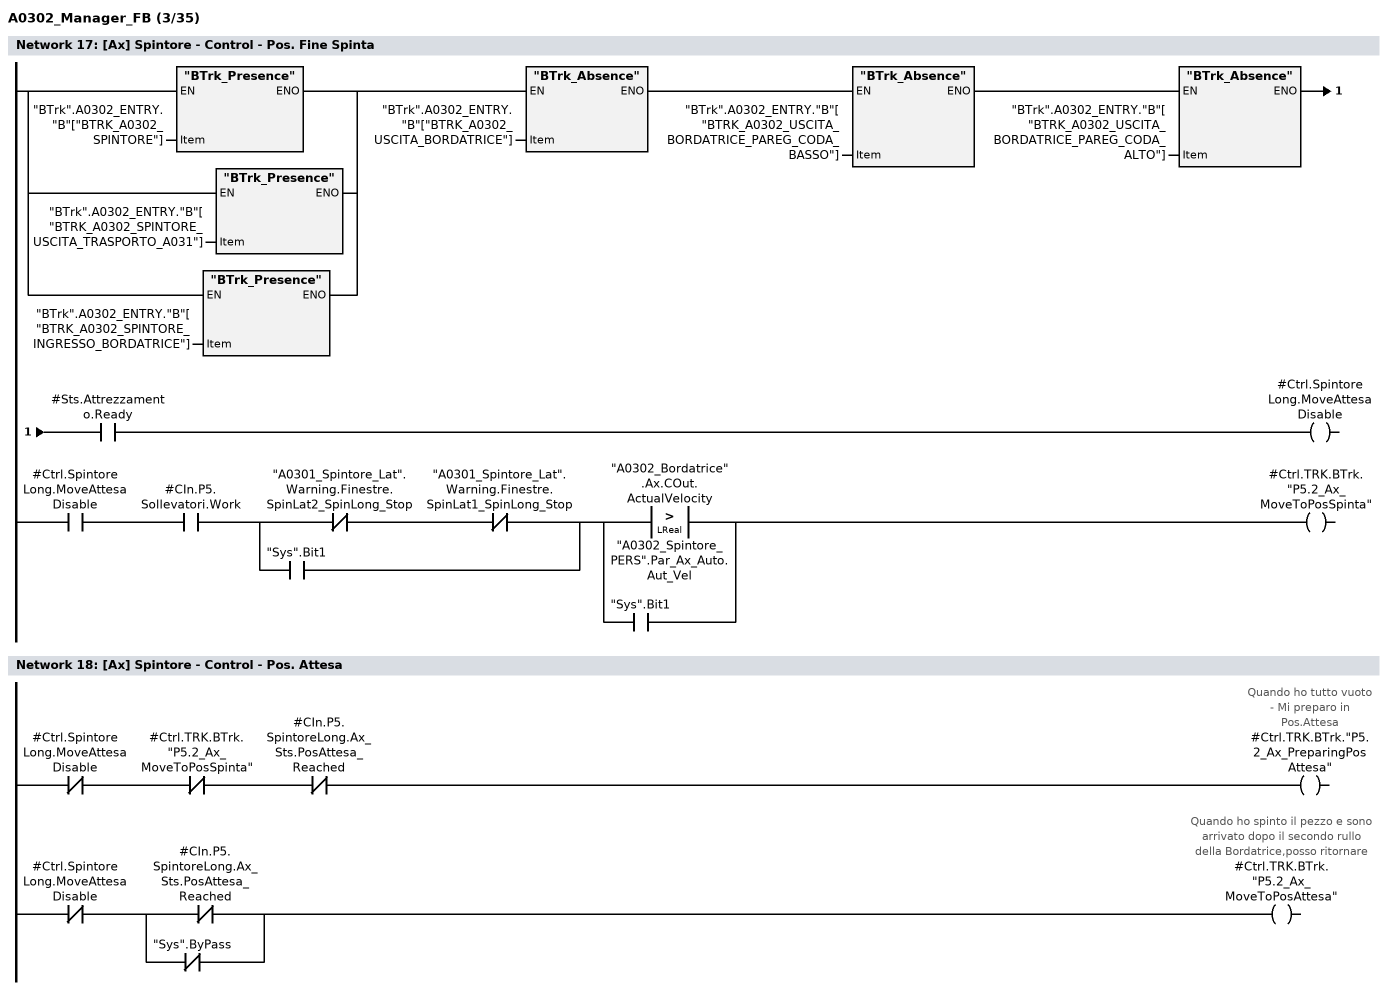
   RUNG wire#powerrail
      "BTrk_Presence"(Item := "BTrk".A0302_ENTRY."B"["BTRK_A0302_SPINTORE"])
      wire#w1
      "BTrk_Absence"(Item := "BTrk".A0302_ENTRY."B"["BTRK_A0302_USCITA_BORDATRICE"])
      "BTrk_Absence"(Item := "BTrk".A0302_ENTRY."B"["BTRK_A0302_USCITA_BORDATRICE_PAREG_CODA_BASSO"])
      "BTrk_Absence"(Item := "BTrk".A0302_ENTRY."B"["BTRK_A0302_USCITA_BORDATRICE_PAREG_CODA_ALTO"])
      Contact( #Sts.Attrezzamento.Ready )
      Coil( #Ctrl.SpintoreLong.MoveAttesaDisable )
   END_RUNG
   RUNG wire#powerrail
      "BTrk_Presence"(Item := "BTrk".A0302_ENTRY."B"["BTRK_A0302_SPINTORE_USCITA_TRASPORTO_A031"])
   END_RUNG wire#w1
   RUNG wire#powerrail
      "BTrk_Presence"(Item := "BTrk".A0302_ENTRY."B"["BTRK_A0302_SPINTORE_INGRESSO_BORDATRICE"])
   END_RUNG wire#w1
   RUNG wire#powerrail
      Contact( #Ctrl.SpintoreLong.MoveAttesaDisable )
      Contact( #CIn.P5.Sollevatori.Work )
      wire#w2
      I_Contact( "A0301_Spintore_Lat".Warning.Finestre.SpinLat2_SpinLong_Stop )
      I_Contact( "A0301_Spintore_Lat".Warning.Finestre.SpinLat1_SpinLong_Stop )
      wire#w3
      { S7_Templates := "SrcType := LReal" } GT_Contact(in1 := "A0302_Bordatrice".Ax.COut.ActualVelocity, in2 := "A0302_Spintore_PERS".Par_Ax_Auto.Aut_Vel)
      wire#w4
      Coil( #Ctrl.TRK.BTrk."P5.2_Ax_MoveToPosSpinta" )
   END_RUNG
   RUNG wire#w2
      Contact( "Sys".Bit1 )
   END_RUNG wire#w3
   RUNG wire#w3
      Contact( "Sys".Bit1 )
   END_RUNG wire#w4
   // the same network as SCL:
   "BTrk_Presence"(Item := "BTrk".A0302_ENTRY."B"["BTRK_A0302_SPINTORE"], ENO => #_w1);
   "BTrk_Presence"(Item := "BTrk".A0302_ENTRY."B"["BTRK_A0302_SPINTORE_USCITA_TRASPORTO_A031"], ENO => #_w2);
   "BTrk_Presence"(Item := "BTrk".A0302_ENTRY."B"["BTRK_A0302_SPINTORE_INGRESSO_BORDATRICE"], ENO => #_w3);
   "BTrk_Absence"(EN := #_w1 OR #_w2 OR #_w3,
                  Item := "BTrk".A0302_ENTRY."B"["BTRK_A0302_USCITA_BORDATRICE"],
                  ENO => #_w4);
   "BTrk_Absence"(EN := #_w4,
                  Item := "BTrk".A0302_ENTRY."B"["BTRK_A0302_USCITA_BORDATRICE_PAREG_CODA_BASSO"],
                  ENO => #_w5);
   "BTrk_Absence"(EN := #_w5,
                  Item := "BTrk".A0302_ENTRY."B"["BTRK_A0302_USCITA_BORDATRICE_PAREG_CODA_ALTO"],
                  ENO => #_w6);
   #Ctrl.SpintoreLong.MoveAttesaDisable := #_w6 AND #Sts.Attrezzamento.Ready;
   #Ctrl.TRK.BTrk."P5.2_Ax_MoveToPosSpinta" := #Ctrl.SpintoreLong.MoveAttesaDisable AND #CIn.P5.Sollevatori.Work AND ((NOT "A0301_Spintore_Lat".Warning.Finestre.SpinLat2_SpinLong_Stop AND NOT "A0301_Spintore_Lat".Warning.Finestre.SpinLat1_SpinLong_Stop) OR "Sys".Bit1) AND (("A0302_Bordatrice".Ax.COut.ActualVelocity > "A0302_Spintore_PERS".Par_Ax_Auto.Aut_Vel) OR "Sys".Bit1);
END_REGION

REGION Network 18: [Ax] Spintore - Control - Pos. Attesa
   RUNG wire#powerrail
      I_Contact( #Ctrl.SpintoreLong.MoveAttesaDisable )
      I_Contact( #Ctrl.TRK.BTrk."P5.2_Ax_MoveToPosSpinta" )
      I_Contact( #CIn.P5.SpintoreLong.Ax_Sts.PosAttesa_Reached )
      Coil( #Ctrl.TRK.BTrk."P5.2_Ax_PreparingPosAttesa" )   // Quando ho tutto vuoto - Mi preparo in Pos.Attesa
   END_RUNG
   RUNG wire#powerrail
      I_Contact( #Ctrl.SpintoreLong.MoveAttesaDisable )
      wire#w1
      I_Contact( #CIn.P5.SpintoreLong.Ax_Sts.PosAttesa_Reached )
      wire#w2
      Coil( #Ctrl.TRK.BTrk."P5.2_Ax_MoveToPosAttesa" )   // Quando ho spinto il pezzo e sono arrivato dopo il secondo rullo della Bordatrice,posso ritornare
   END_RUNG
   RUNG wire#w1
      I_Contact( "Sys".ByPass )
   END_RUNG wire#w2
   // the same network as SCL:
   #Ctrl.TRK.BTrk."P5.2_Ax_PreparingPosAttesa" := NOT #Ctrl.SpintoreLong.MoveAttesaDisable AND NOT #Ctrl.TRK.BTrk."P5.2_Ax_MoveToPosSpinta" AND NOT #CIn.P5.SpintoreLong.Ax_Sts.PosAttesa_Reached;   // Quando ho tutto vuoto - Mi preparo in Pos.Attesa
   #Ctrl.TRK.BTrk."P5.2_Ax_MoveToPosAttesa" := NOT #Ctrl.SpintoreLong.MoveAttesaDisable AND (NOT #CIn.P5.SpintoreLong.Ax_Sts.PosAttesa_Reached OR NOT "Sys".ByPass);   // Quando ho spinto il pezzo e sono arrivato dopo il secondo rullo della Bordatrice,posso ritornare
END_REGION

REGION Network 19: [Ax] Spintore Longitudinale - COut Manager
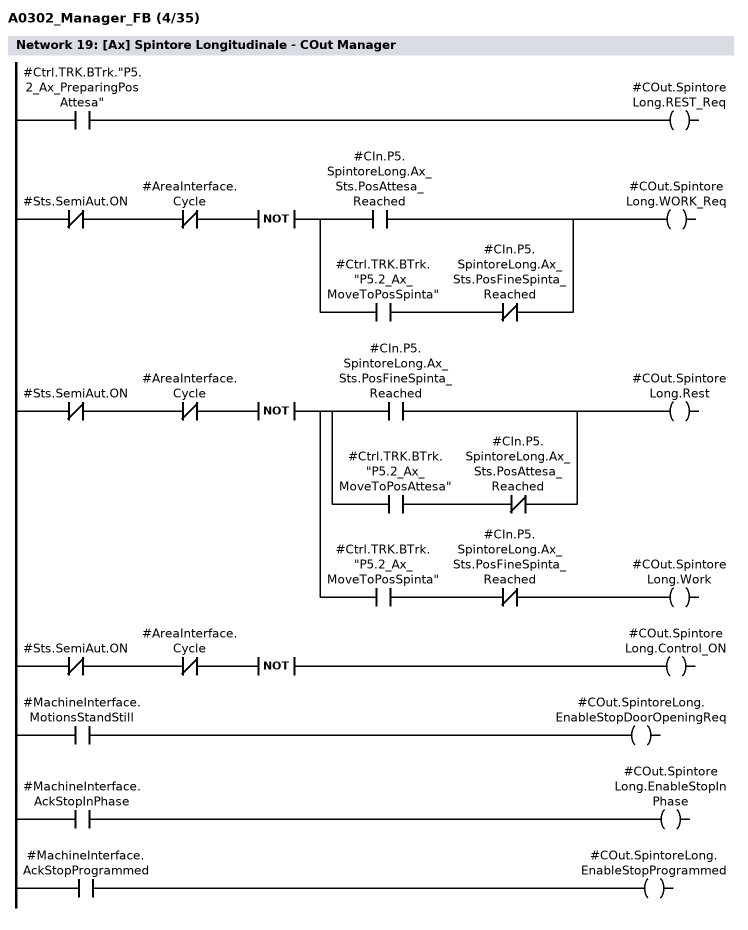
   RUNG wire#powerrail
      Contact( #Ctrl.TRK.BTrk."P5.2_Ax_PreparingPosAttesa" )
      Coil( #COut.SpintoreLong.REST_Req )
   END_RUNG
   RUNG wire#powerrail
      I_Contact( #Sts.SemiAut.ON )
      I_Contact( #AreaInterface.Cycle )
      Not()
      wire#w1
      Contact( #CIn.P5.SpintoreLong.Ax_Sts.PosAttesa_Reached )
      wire#w2
      Coil( #COut.SpintoreLong.WORK_Req )
   END_RUNG
   RUNG wire#w1
      Contact( #Ctrl.TRK.BTrk."P5.2_Ax_MoveToPosSpinta" )
      I_Contact( #CIn.P5.SpintoreLong.Ax_Sts.PosFineSpinta_Reached )
   END_RUNG wire#w2
   RUNG wire#powerrail
      I_Contact( #Sts.SemiAut.ON )
      I_Contact( #AreaInterface.Cycle )
      Not()
      wire#w3
      Contact( #CIn.P5.SpintoreLong.Ax_Sts.PosFineSpinta_Reached )
      wire#w4
      Coil( #COut.SpintoreLong.Rest )
   END_RUNG
   RUNG wire#w3
      Contact( #Ctrl.TRK.BTrk."P5.2_Ax_MoveToPosAttesa" )
      I_Contact( #CIn.P5.SpintoreLong.Ax_Sts.PosAttesa_Reached )
   END_RUNG wire#w4
   RUNG wire#w3
      Contact( #Ctrl.TRK.BTrk."P5.2_Ax_MoveToPosSpinta" )
      I_Contact( #CIn.P5.SpintoreLong.Ax_Sts.PosFineSpinta_Reached )
      Coil( #COut.SpintoreLong.Work )
   END_RUNG
   RUNG wire#powerrail
      I_Contact( #Sts.SemiAut.ON )
      I_Contact( #AreaInterface.Cycle )
      Not()
      Coil( #COut.SpintoreLong.Control_ON )
   END_RUNG
   RUNG wire#powerrail
      Contact( #MachineInterface.MotionsStandStill )
      Coil( #COut.SpintoreLong.EnableStopDoorOpeningReq )
   END_RUNG
   RUNG wire#powerrail
      Contact( #MachineInterface.AckStopInPhase )
      Coil( #COut.SpintoreLong.EnableStopInPhase )
   END_RUNG
   RUNG wire#powerrail
      Contact( #MachineInterface.AckStopProgrammed )
      Coil( #COut.SpintoreLong.EnableStopProgrammed )
   END_RUNG
   // the same network as SCL:
   #COut.SpintoreLong.REST_Req := #Ctrl.TRK.BTrk."P5.2_Ax_PreparingPosAttesa";
   #COut.SpintoreLong.WORK_Req := NOT (NOT #Sts.SemiAut.ON AND NOT #AreaInterface.Cycle) AND (#CIn.P5.SpintoreLong.Ax_Sts.PosAttesa_Reached OR (#Ctrl.TRK.BTrk."P5.2_Ax_MoveToPosSpinta" AND NOT #CIn.P5.SpintoreLong.Ax_Sts.PosFineSpinta_Reached));
   #_w1 := NOT (NOT #Sts.SemiAut.ON AND NOT #AreaInterface.Cycle);
   #COut.SpintoreLong.Rest := #_w1 AND (#CIn.P5.SpintoreLong.Ax_Sts.PosFineSpinta_Reached OR (#Ctrl.TRK.BTrk."P5.2_Ax_MoveToPosAttesa" AND NOT #CIn.P5.SpintoreLong.Ax_Sts.PosAttesa_Reached));
   #COut.SpintoreLong.Work := #_w1 AND #Ctrl.TRK.BTrk."P5.2_Ax_MoveToPosSpinta" AND NOT #CIn.P5.SpintoreLong.Ax_Sts.PosFineSpinta_Reached;
   #COut.SpintoreLong.Control_ON := NOT (NOT #Sts.SemiAut.ON AND NOT #AreaInterface.Cycle);
   #COut.SpintoreLong.EnableStopDoorOpeningReq := #MachineInterface.MotionsStandStill;
   #COut.SpintoreLong.EnableStopInPhase := #MachineInterface.AckStopInPhase;
   #COut.SpintoreLong.EnableStopProgrammed := #MachineInterface.AckStopProgrammed;
END_REGION

REGION Network 21: <<<< BORDATRICE >>>>
END_REGION

REGION Network 22: [Ax] Movimento BTrk Spin Ingresso Bordatrice ==a==> Ingresso Bordatrice
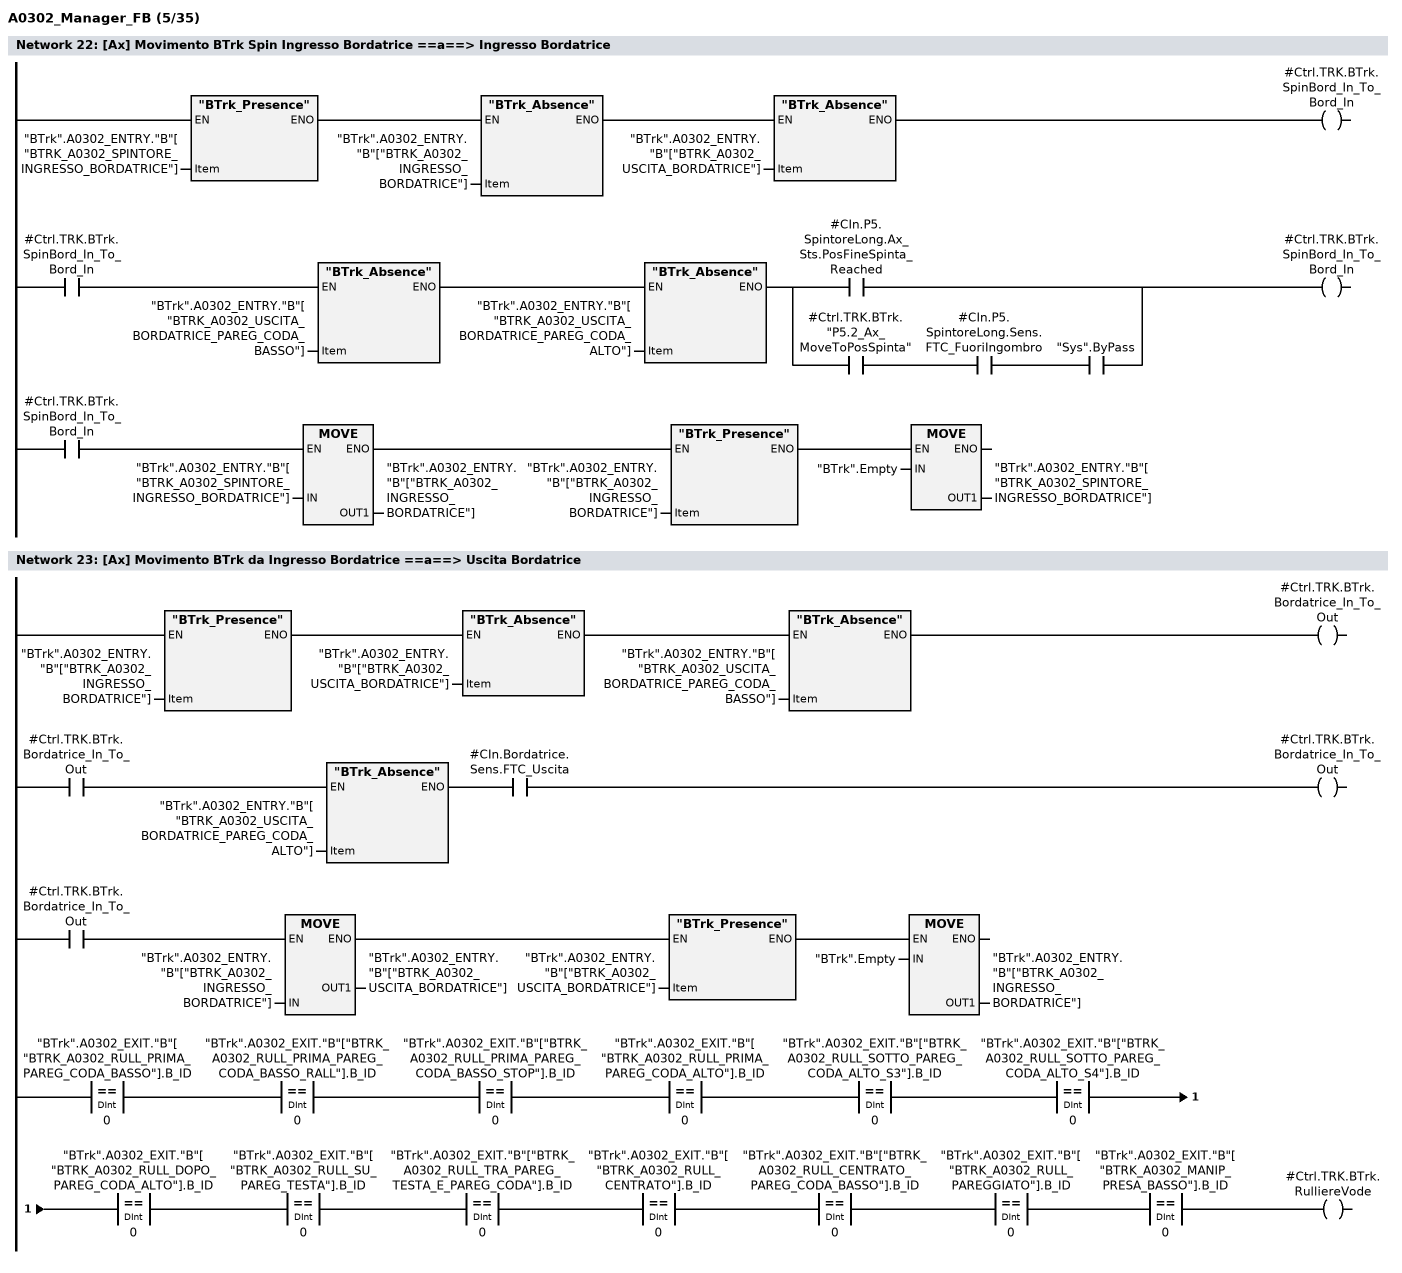
   RUNG wire#powerrail
      "BTrk_Presence"(Item := "BTrk".A0302_ENTRY."B"["BTRK_A0302_SPINTORE_INGRESSO_BORDATRICE"])
      "BTrk_Absence"(Item := "BTrk".A0302_ENTRY."B"["BTRK_A0302_INGRESSO_BORDATRICE"])
      "BTrk_Absence"(Item := "BTrk".A0302_ENTRY."B"["BTRK_A0302_USCITA_BORDATRICE"])
      Coil( #Ctrl.TRK.BTrk.SpinBord_In_To_Bord_In )
   END_RUNG
   RUNG wire#powerrail
      Contact( #Ctrl.TRK.BTrk.SpinBord_In_To_Bord_In )
      "BTrk_Absence"(Item := "BTrk".A0302_ENTRY."B"["BTRK_A0302_USCITA_BORDATRICE_PAREG_CODA_BASSO"])
      "BTrk_Absence"(Item := "BTrk".A0302_ENTRY."B"["BTRK_A0302_USCITA_BORDATRICE_PAREG_CODA_ALTO"])
      wire#w1
      Contact( #CIn.P5.SpintoreLong.Ax_Sts.PosFineSpinta_Reached )
      wire#w2
      Coil( #Ctrl.TRK.BTrk.SpinBord_In_To_Bord_In )
   END_RUNG
   RUNG wire#w1
      Contact( #Ctrl.TRK.BTrk."P5.2_Ax_MoveToPosSpinta" )
      Contact( #CIn.P5.SpintoreLong.Sens.FTC_FuoriIngombro )
      Contact( "Sys".ByPass )
   END_RUNG wire#w2
   RUNG wire#powerrail
      Contact( #Ctrl.TRK.BTrk.SpinBord_In_To_Bord_In )
      Move(in := "BTrk".A0302_ENTRY."B"["BTRK_A0302_SPINTORE_INGRESSO_BORDATRICE"], out1 => "BTrk".A0302_ENTRY."B"["BTRK_A0302_INGRESSO_BORDATRICE"])
      "BTrk_Presence"(Item := "BTrk".A0302_ENTRY."B"["BTRK_A0302_INGRESSO_BORDATRICE"])
      Move(in := "BTrk".Empty, out1 => "BTrk".A0302_ENTRY."B"["BTRK_A0302_SPINTORE_INGRESSO_BORDATRICE"])
   END_RUNG
   // the same network as SCL:
   "BTrk_Presence"(Item := "BTrk".A0302_ENTRY."B"["BTRK_A0302_SPINTORE_INGRESSO_BORDATRICE"], ENO => #_w1);
   "BTrk_Absence"(EN := #_w1, Item := "BTrk".A0302_ENTRY."B"["BTRK_A0302_INGRESSO_BORDATRICE"], ENO => #_w2);
   "BTrk_Absence"(EN := #_w2, Item := "BTrk".A0302_ENTRY."B"["BTRK_A0302_USCITA_BORDATRICE"], ENO => #_w3);
   #Ctrl.TRK.BTrk.SpinBord_In_To_Bord_In := #_w3;
   "BTrk_Absence"(EN := #Ctrl.TRK.BTrk.SpinBord_In_To_Bord_In,
                  Item := "BTrk".A0302_ENTRY."B"["BTRK_A0302_USCITA_BORDATRICE_PAREG_CODA_BASSO"],
                  ENO => #_w4);
   "BTrk_Absence"(EN := #_w4,
                  Item := "BTrk".A0302_ENTRY."B"["BTRK_A0302_USCITA_BORDATRICE_PAREG_CODA_ALTO"],
                  ENO => #_w5);
   #Ctrl.TRK.BTrk.SpinBord_In_To_Bord_In := #_w5 AND (#CIn.P5.SpintoreLong.Ax_Sts.PosFineSpinta_Reached OR (#Ctrl.TRK.BTrk."P5.2_Ax_MoveToPosSpinta" AND #CIn.P5.SpintoreLong.Sens.FTC_FuoriIngombro AND "Sys".ByPass));
   IF #Ctrl.TRK.BTrk.SpinBord_In_To_Bord_In THEN
       "BTrk".A0302_ENTRY."B"["BTRK_A0302_INGRESSO_BORDATRICE"] := "BTrk".A0302_ENTRY."B"["BTRK_A0302_SPINTORE_INGRESSO_BORDATRICE"];
   END_IF;
   "BTrk_Presence"(EN := #Ctrl.TRK.BTrk.SpinBord_In_To_Bord_In,
                   Item := "BTrk".A0302_ENTRY."B"["BTRK_A0302_INGRESSO_BORDATRICE"],
                   ENO => #_w6);
   IF #_w6 THEN "BTrk".A0302_ENTRY."B"["BTRK_A0302_SPINTORE_INGRESSO_BORDATRICE"] := "BTrk".Empty; END_IF;
END_REGION

REGION Network 23: [Ax] Movimento BTrk da Ingresso Bordatrice ==a==> Uscita Bordatrice
   RUNG wire#powerrail
      "BTrk_Presence"(Item := "BTrk".A0302_ENTRY."B"["BTRK_A0302_INGRESSO_BORDATRICE"])
      "BTrk_Absence"(Item := "BTrk".A0302_ENTRY."B"["BTRK_A0302_USCITA_BORDATRICE"])
      "BTrk_Absence"(Item := "BTrk".A0302_ENTRY."B"["BTRK_A0302_USCITA_BORDATRICE_PAREG_CODA_BASSO"])
      Coil( #Ctrl.TRK.BTrk.Bordatrice_In_To_Out )
   END_RUNG
   RUNG wire#powerrail
      Contact( #Ctrl.TRK.BTrk.Bordatrice_In_To_Out )
      "BTrk_Absence"(Item := "BTrk".A0302_ENTRY."B"["BTRK_A0302_USCITA_BORDATRICE_PAREG_CODA_ALTO"])
      Contact( #CIn.Bordatrice.Sens.FTC_Uscita )
      Coil( #Ctrl.TRK.BTrk.Bordatrice_In_To_Out )
   END_RUNG
   RUNG wire#powerrail
      Contact( #Ctrl.TRK.BTrk.Bordatrice_In_To_Out )
      Move(in := "BTrk".A0302_ENTRY."B"["BTRK_A0302_INGRESSO_BORDATRICE"], out1 => "BTrk".A0302_ENTRY."B"["BTRK_A0302_USCITA_BORDATRICE"])
      "BTrk_Presence"(Item := "BTrk".A0302_ENTRY."B"["BTRK_A0302_USCITA_BORDATRICE"])
      Move(in := "BTrk".Empty, out1 => "BTrk".A0302_ENTRY."B"["BTRK_A0302_INGRESSO_BORDATRICE"])
   END_RUNG
   RUNG wire#powerrail
      { S7_Templates := "SrcType := DInt" } EQ_Contact(in1 := "BTrk".A0302_EXIT."B"["BTRK_A0302_RULL_PRIMA_PAREG_CODA_BASSO"].B_ID, in2 := 0)
      { S7_Templates := "SrcType := DInt" } EQ_Contact(in1 := "BTrk".A0302_EXIT."B"["BTRK_A0302_RULL_PRIMA_PAREG_CODA_BASSO_RALL"].B_ID, in2 := 0)
      { S7_Templates := "SrcType := DInt" } EQ_Contact(in1 := "BTrk".A0302_EXIT."B"["BTRK_A0302_RULL_PRIMA_PAREG_CODA_BASSO_STOP"].B_ID, in2 := 0)
      { S7_Templates := "SrcType := DInt" } EQ_Contact(in1 := "BTrk".A0302_EXIT."B"["BTRK_A0302_RULL_PRIMA_PAREG_CODA_ALTO"].B_ID, in2 := 0)
      { S7_Templates := "SrcType := DInt" } EQ_Contact(in1 := "BTrk".A0302_EXIT."B"["BTRK_A0302_RULL_SOTTO_PAREG_CODA_ALTO_S3"].B_ID, in2 := 0)
      { S7_Templates := "SrcType := DInt" } EQ_Contact(in1 := "BTrk".A0302_EXIT."B"["BTRK_A0302_RULL_SOTTO_PAREG_CODA_ALTO_S4"].B_ID, in2 := 0)
      { S7_Templates := "SrcType := DInt" } EQ_Contact(in1 := "BTrk".A0302_EXIT."B"["BTRK_A0302_RULL_DOPO_PAREG_CODA_ALTO"].B_ID, in2 := 0)
      { S7_Templates := "SrcType := DInt" } EQ_Contact(in1 := "BTrk".A0302_EXIT."B"["BTRK_A0302_RULL_SU_PAREG_TESTA"].B_ID, in2 := 0)
      { S7_Templates := "SrcType := DInt" } EQ_Contact(in1 := "BTrk".A0302_EXIT."B"["BTRK_A0302_RULL_TRA_PAREG_TESTA_E_PAREG_CODA"].B_ID, in2 := 0)
      { S7_Templates := "SrcType := DInt" } EQ_Contact(in1 := "BTrk".A0302_EXIT."B"["BTRK_A0302_RULL_CENTRATO"].B_ID, in2 := 0)
      { S7_Templates := "SrcType := DInt" } EQ_Contact(in1 := "BTrk".A0302_EXIT."B"["BTRK_A0302_RULL_CENTRATO_PAREG_CODA_BASSO"].B_ID, in2 := 0)
      { S7_Templates := "SrcType := DInt" } EQ_Contact(in1 := "BTrk".A0302_EXIT."B"["BTRK_A0302_RULL_PAREGGIATO"].B_ID, in2 := 0)
      { S7_Templates := "SrcType := DInt" } EQ_Contact(in1 := "BTrk".A0302_EXIT."B"["BTRK_A0302_MANIP_PRESA_BASSO"].B_ID, in2 := 0)
      Coil( #Ctrl.TRK.BTrk.RulliereVode )
   END_RUNG
   // the same network as SCL:
   "BTrk_Presence"(Item := "BTrk".A0302_ENTRY."B"["BTRK_A0302_INGRESSO_BORDATRICE"], ENO => #_w1);
   "BTrk_Absence"(EN := #_w1, Item := "BTrk".A0302_ENTRY."B"["BTRK_A0302_USCITA_BORDATRICE"], ENO => #_w2);
   "BTrk_Absence"(EN := #_w2,
                  Item := "BTrk".A0302_ENTRY."B"["BTRK_A0302_USCITA_BORDATRICE_PAREG_CODA_BASSO"],
                  ENO => #_w3);
   #Ctrl.TRK.BTrk.Bordatrice_In_To_Out := #_w3;
   "BTrk_Absence"(EN := #Ctrl.TRK.BTrk.Bordatrice_In_To_Out,
                  Item := "BTrk".A0302_ENTRY."B"["BTRK_A0302_USCITA_BORDATRICE_PAREG_CODA_ALTO"],
                  ENO => #_w4);
   #Ctrl.TRK.BTrk.Bordatrice_In_To_Out := #_w4 AND #CIn.Bordatrice.Sens.FTC_Uscita;
   IF #Ctrl.TRK.BTrk.Bordatrice_In_To_Out THEN
       "BTrk".A0302_ENTRY."B"["BTRK_A0302_USCITA_BORDATRICE"] := "BTrk".A0302_ENTRY."B"["BTRK_A0302_INGRESSO_BORDATRICE"];
   END_IF;
   "BTrk_Presence"(EN := #Ctrl.TRK.BTrk.Bordatrice_In_To_Out,
                   Item := "BTrk".A0302_ENTRY."B"["BTRK_A0302_USCITA_BORDATRICE"],
                   ENO => #_w5);
   IF #_w5 THEN "BTrk".A0302_ENTRY."B"["BTRK_A0302_INGRESSO_BORDATRICE"] := "BTrk".Empty; END_IF;
   #Ctrl.TRK.BTrk.RulliereVode := ("BTrk".A0302_EXIT."B"["BTRK_A0302_RULL_PRIMA_PAREG_CODA_BASSO"].B_ID = 0) AND ("BTrk".A0302_EXIT."B"["BTRK_A0302_RULL_PRIMA_PAREG_CODA_BASSO_RALL"].B_ID = 0) AND ("BTrk".A0302_EXIT."B"["BTRK_A0302_RULL_PRIMA_PAREG_CODA_BASSO_STOP"].B_ID = 0) AND ("BTrk".A0302_EXIT."B"["BTRK_A0302_RULL_PRIMA_PAREG_CODA_ALTO"].B_ID = 0) AND ("BTrk".A0302_EXIT."B"["BTRK_A0302_RULL_SOTTO_PAREG_CODA_ALTO_S3"].B_ID = 0) AND ("BTrk".A0302_EXIT."B"["BTRK_A0302_RULL_SOTTO_PAREG_CODA_ALTO_S4"].B_ID = 0) AND ("BTrk".A0302_EXIT."B"["BTRK_A0302_RULL_DOPO_PAREG_CODA_ALTO"].B_ID = 0) AND ("BTrk".A0302_EXIT."B"["BTRK_A0302_RULL_SU_PAREG_TESTA"].B_ID = 0) AND ("BTrk".A0302_EXIT."B"["BTRK_A0302_RULL_TRA_PAREG_TESTA_E_PAREG_CODA"].B_ID = 0) AND ("BTrk".A0302_EXIT."B"["BTRK_A0302_RULL_CENTRATO"].B_ID = 0) AND ("BTrk".A0302_EXIT."B"["BTRK_A0302_RULL_CENTRATO_PAREG_CODA_BASSO"].B_ID = 0) AND ("BTrk".A0302_EXIT."B"["BTRK_A0302_RULL_PAREGGIATO"].B_ID = 0) AND ("BTrk".A0302_EXIT."B"["BTRK_A0302_MANIP_PRESA_BASSO"].B_ID = 0);
END_REGION

REGION Network 24: [Ax] Movimento BTrk da Uscita Bordatrice ==a==> Uscita Bord. Pareggiatore Coda Basso
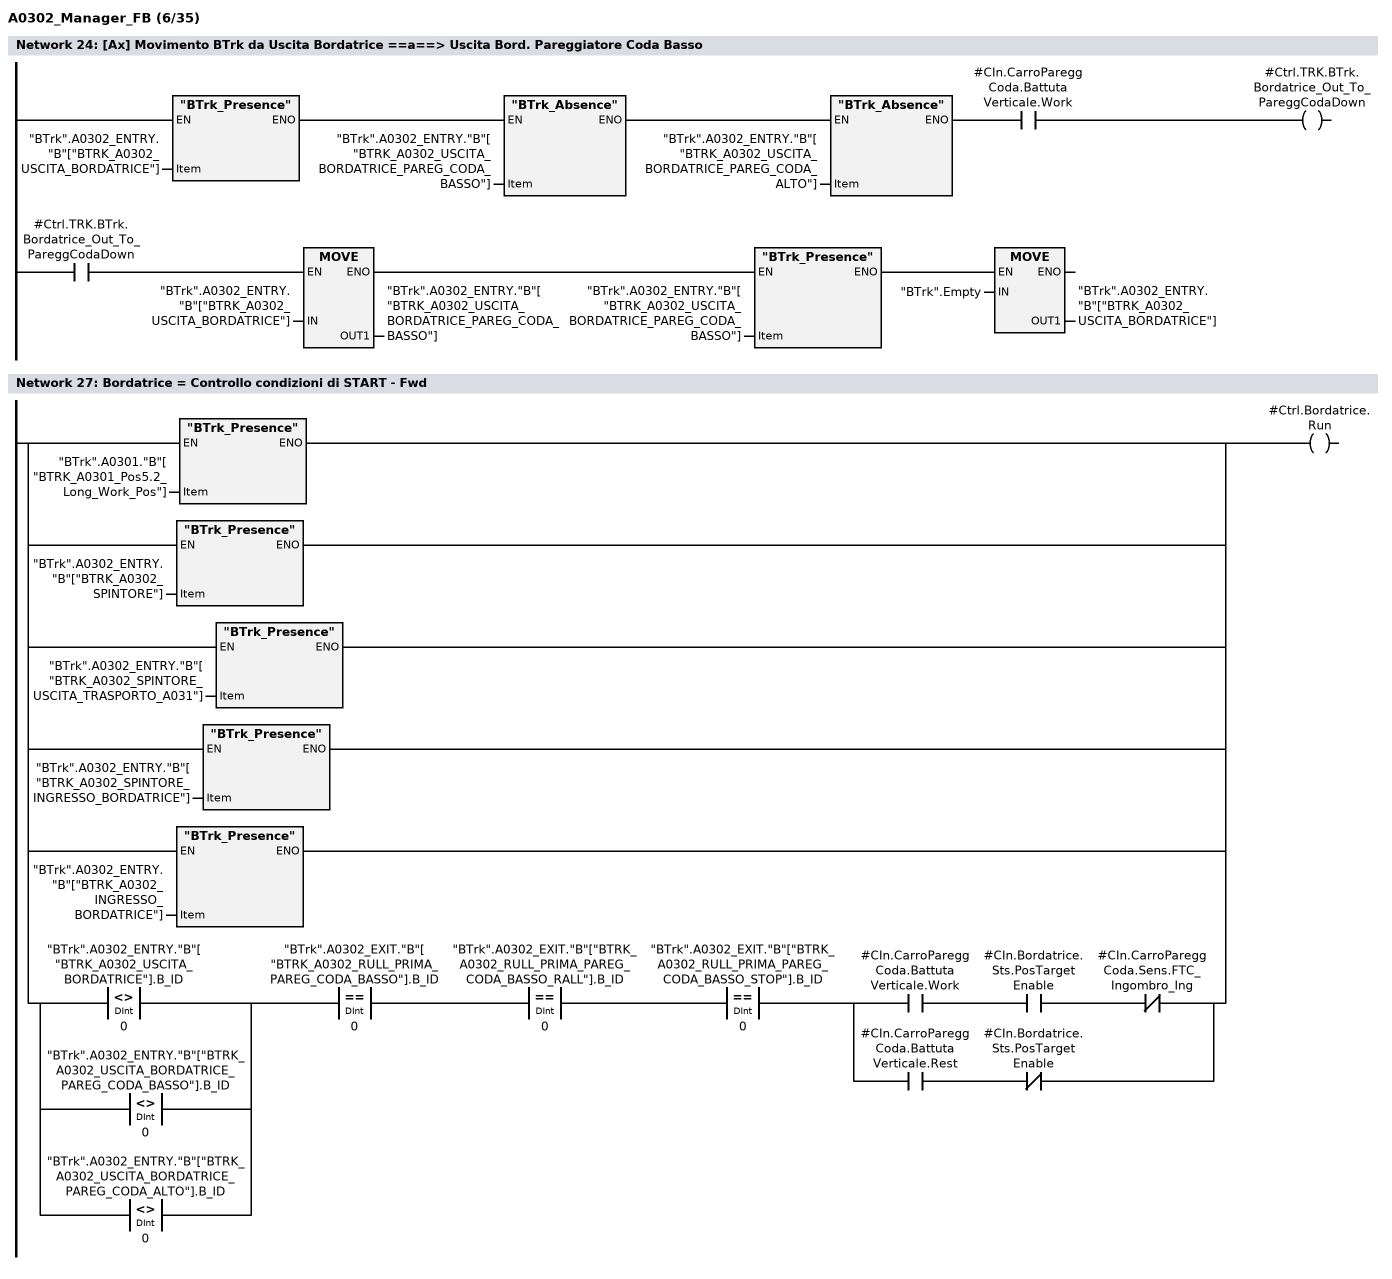
   RUNG wire#powerrail
      "BTrk_Presence"(Item := "BTrk".A0302_ENTRY."B"["BTRK_A0302_USCITA_BORDATRICE"])
      "BTrk_Absence"(Item := "BTrk".A0302_ENTRY."B"["BTRK_A0302_USCITA_BORDATRICE_PAREG_CODA_BASSO"])
      "BTrk_Absence"(Item := "BTrk".A0302_ENTRY."B"["BTRK_A0302_USCITA_BORDATRICE_PAREG_CODA_ALTO"])
      Contact( #CIn.CarroPareggCoda.BattutaVerticale.Work )
      Coil( #Ctrl.TRK.BTrk.Bordatrice_Out_To_PareggCodaDown )
   END_RUNG
   RUNG wire#powerrail
      Contact( #Ctrl.TRK.BTrk.Bordatrice_Out_To_PareggCodaDown )
      Move(in := "BTrk".A0302_ENTRY."B"["BTRK_A0302_USCITA_BORDATRICE"], out1 => "BTrk".A0302_ENTRY."B"["BTRK_A0302_USCITA_BORDATRICE_PAREG_CODA_BASSO"])
      "BTrk_Presence"(Item := "BTrk".A0302_ENTRY."B"["BTRK_A0302_USCITA_BORDATRICE_PAREG_CODA_BASSO"])
      Move(in := "BTrk".Empty, out1 => "BTrk".A0302_ENTRY."B"["BTRK_A0302_USCITA_BORDATRICE"])
   END_RUNG
   // the same network as SCL:
   "BTrk_Presence"(Item := "BTrk".A0302_ENTRY."B"["BTRK_A0302_USCITA_BORDATRICE"], ENO => #_w1);
   "BTrk_Absence"(EN := #_w1,
                  Item := "BTrk".A0302_ENTRY."B"["BTRK_A0302_USCITA_BORDATRICE_PAREG_CODA_BASSO"],
                  ENO => #_w2);
   "BTrk_Absence"(EN := #_w2,
                  Item := "BTrk".A0302_ENTRY."B"["BTRK_A0302_USCITA_BORDATRICE_PAREG_CODA_ALTO"],
                  ENO => #_w3);
   #Ctrl.TRK.BTrk.Bordatrice_Out_To_PareggCodaDown := #_w3 AND #CIn.CarroPareggCoda.BattutaVerticale.Work;
   IF #Ctrl.TRK.BTrk.Bordatrice_Out_To_PareggCodaDown THEN
       "BTrk".A0302_ENTRY."B"["BTRK_A0302_USCITA_BORDATRICE_PAREG_CODA_BASSO"] := "BTrk".A0302_ENTRY."B"["BTRK_A0302_USCITA_BORDATRICE"];
   END_IF;
   "BTrk_Presence"(EN := #Ctrl.TRK.BTrk.Bordatrice_Out_To_PareggCodaDown,
                   Item := "BTrk".A0302_ENTRY."B"["BTRK_A0302_USCITA_BORDATRICE_PAREG_CODA_BASSO"],
                   ENO => #_w4);
   IF #_w4 THEN "BTrk".A0302_ENTRY."B"["BTRK_A0302_USCITA_BORDATRICE"] := "BTrk".Empty; END_IF;
END_REGION

REGION Network 26: <<<< GESTIONE MOVIMENTO BORDATRICE >>>>
END_REGION

REGION Network 27: Bordatrice = Controllo condizioni di START - Fwd
   RUNG wire#powerrail
      "BTrk_Presence"(Item := "BTrk".A0301."B"["BTRK_A0301_Pos5.2_Long_Work_Pos"])
      wire#w1
      Coil( #Ctrl.Bordatrice.Run )
   END_RUNG
   RUNG wire#powerrail
      "BTrk_Presence"(Item := "BTrk".A0302_ENTRY."B"["BTRK_A0302_SPINTORE"])
   END_RUNG wire#w1
   RUNG wire#powerrail
      "BTrk_Presence"(Item := "BTrk".A0302_ENTRY."B"["BTRK_A0302_SPINTORE_USCITA_TRASPORTO_A031"])
   END_RUNG wire#w1
   RUNG wire#powerrail
      "BTrk_Presence"(Item := "BTrk".A0302_ENTRY."B"["BTRK_A0302_SPINTORE_INGRESSO_BORDATRICE"])
   END_RUNG wire#w1
   RUNG wire#powerrail
      "BTrk_Presence"(Item := "BTrk".A0302_ENTRY."B"["BTRK_A0302_INGRESSO_BORDATRICE"])
   END_RUNG wire#w1
   RUNG wire#powerrail
      { S7_Templates := "SrcType := DInt" } NE_Contact(in1 := "BTrk".A0302_ENTRY."B"["BTRK_A0302_USCITA_BORDATRICE"].B_ID, in2 := 0)
      wire#w2
      { S7_Templates := "SrcType := DInt" } EQ_Contact(in1 := "BTrk".A0302_EXIT."B"["BTRK_A0302_RULL_PRIMA_PAREG_CODA_BASSO"].B_ID, in2 := 0)
      { S7_Templates := "SrcType := DInt" } EQ_Contact(in1 := "BTrk".A0302_EXIT."B"["BTRK_A0302_RULL_PRIMA_PAREG_CODA_BASSO_RALL"].B_ID, in2 := 0)
      { S7_Templates := "SrcType := DInt" } EQ_Contact(in1 := "BTrk".A0302_EXIT."B"["BTRK_A0302_RULL_PRIMA_PAREG_CODA_BASSO_STOP"].B_ID, in2 := 0)
      wire#w3
      Contact( #CIn.CarroPareggCoda.BattutaVerticale.Work )
      Contact( #CIn.Bordatrice.Sts.PosTargetEnable )
      I_Contact( #CIn.CarroPareggCoda.Sens.FTC_Ingombro_Ing )
   END_RUNG wire#w1
   RUNG wire#powerrail
      { S7_Templates := "SrcType := DInt" } NE_Contact(in1 := "BTrk".A0302_ENTRY."B"["BTRK_A0302_USCITA_BORDATRICE_PAREG_CODA_BASSO"].B_ID, in2 := 0)
   END_RUNG wire#w2
   RUNG wire#powerrail
      { S7_Templates := "SrcType := DInt" } NE_Contact(in1 := "BTrk".A0302_ENTRY."B"["BTRK_A0302_USCITA_BORDATRICE_PAREG_CODA_ALTO"].B_ID, in2 := 0)
   END_RUNG wire#w2
   RUNG wire#w3
      Contact( #CIn.CarroPareggCoda.BattutaVerticale.Rest )
      I_Contact( #CIn.Bordatrice.Sts.PosTargetEnable )
   END_RUNG wire#w1
   // the same network as SCL:
   "BTrk_Presence"(Item := "BTrk".A0301."B"["BTRK_A0301_Pos5.2_Long_Work_Pos"], ENO => #_w1);
   "BTrk_Presence"(Item := "BTrk".A0302_ENTRY."B"["BTRK_A0302_SPINTORE"], ENO => #_w2);
   "BTrk_Presence"(Item := "BTrk".A0302_ENTRY."B"["BTRK_A0302_SPINTORE_USCITA_TRASPORTO_A031"], ENO => #_w3);
   "BTrk_Presence"(Item := "BTrk".A0302_ENTRY."B"["BTRK_A0302_SPINTORE_INGRESSO_BORDATRICE"], ENO => #_w4);
   "BTrk_Presence"(Item := "BTrk".A0302_ENTRY."B"["BTRK_A0302_INGRESSO_BORDATRICE"], ENO => #_w5);
   #Ctrl.Bordatrice.Run := #_w1 OR #_w2 OR #_w3 OR #_w4 OR #_w5 OR ((("BTrk".A0302_ENTRY."B"["BTRK_A0302_USCITA_BORDATRICE"].B_ID <> 0) OR ("BTrk".A0302_ENTRY."B"["BTRK_A0302_USCITA_BORDATRICE_PAREG_CODA_BASSO"].B_ID <> 0) OR ("BTrk".A0302_ENTRY."B"["BTRK_A0302_USCITA_BORDATRICE_PAREG_CODA_ALTO"].B_ID <> 0)) AND ("BTrk".A0302_EXIT."B"["BTRK_A0302_RULL_PRIMA_PAREG_CODA_BASSO"].B_ID = 0) AND ("BTrk".A0302_EXIT."B"["BTRK_A0302_RULL_PRIMA_PAREG_CODA_BASSO_RALL"].B_ID = 0) AND ("BTrk".A0302_EXIT."B"["BTRK_A0302_RULL_PRIMA_PAREG_CODA_BASSO_STOP"].B_ID = 0) AND ((#CIn.CarroPareggCoda.BattutaVerticale.Work AND #CIn.Bordatrice.Sts.PosTargetEnable AND NOT #CIn.CarroPareggCoda.Sens.FTC_Ingombro_Ing) OR (#CIn.CarroPareggCoda.BattutaVerticale.Rest AND NOT #CIn.Bordatrice.Sts.PosTargetEnable)));
END_REGION

REGION Network 28: [Ax] Bordatrice = COut Manager
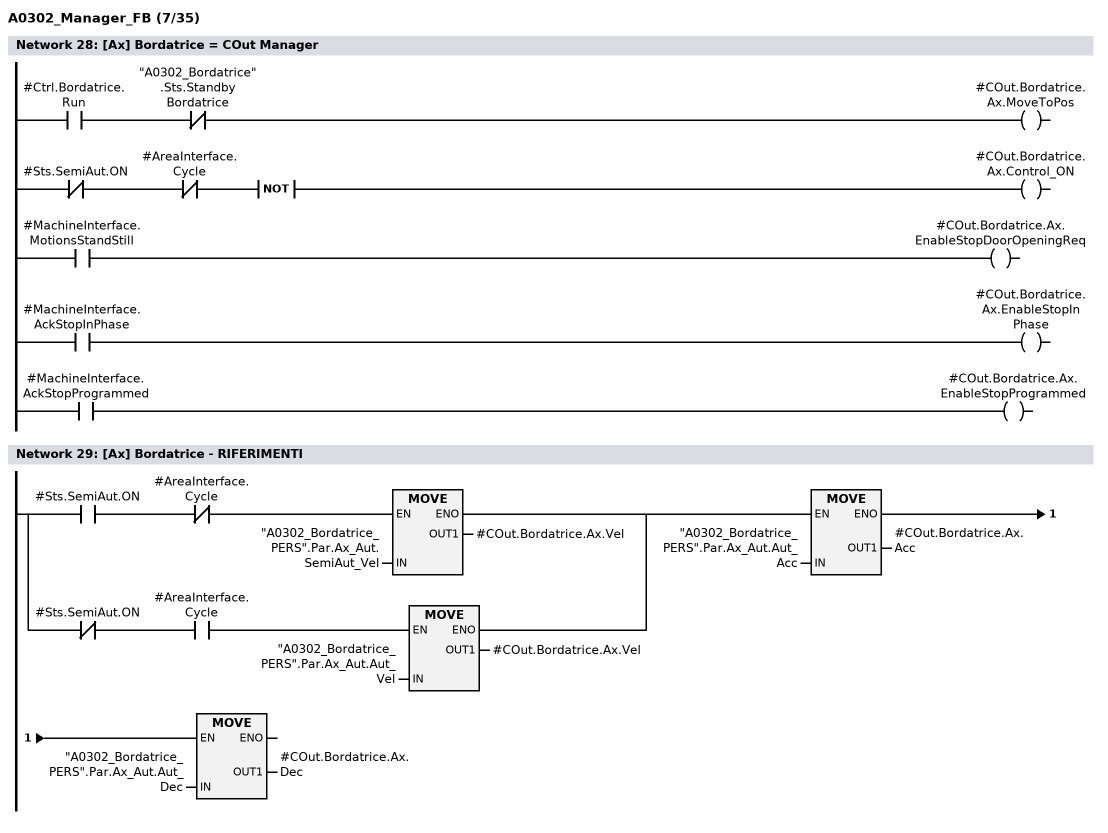
   RUNG wire#powerrail
      Contact( #Ctrl.Bordatrice.Run )
      I_Contact( "A0302_Bordatrice".Sts.StandbyBordatrice )
      Coil( #COut.Bordatrice.Ax.MoveToPos )
   END_RUNG
   RUNG wire#powerrail
      I_Contact( #Sts.SemiAut.ON )
      I_Contact( #AreaInterface.Cycle )
      Not()
      Coil( #COut.Bordatrice.Ax.Control_ON )
   END_RUNG
   RUNG wire#powerrail
      Contact( #MachineInterface.MotionsStandStill )
      Coil( #COut.Bordatrice.Ax.EnableStopDoorOpeningReq )
   END_RUNG
   RUNG wire#powerrail
      Contact( #MachineInterface.AckStopInPhase )
      Coil( #COut.Bordatrice.Ax.EnableStopInPhase )
   END_RUNG
   RUNG wire#powerrail
      Contact( #MachineInterface.AckStopProgrammed )
      Coil( #COut.Bordatrice.Ax.EnableStopProgrammed )
   END_RUNG
   // the same network as SCL:
   #COut.Bordatrice.Ax.MoveToPos := #Ctrl.Bordatrice.Run AND NOT "A0302_Bordatrice".Sts.StandbyBordatrice;
   #COut.Bordatrice.Ax.Control_ON := NOT (NOT #Sts.SemiAut.ON AND NOT #AreaInterface.Cycle);
   #COut.Bordatrice.Ax.EnableStopDoorOpeningReq := #MachineInterface.MotionsStandStill;
   #COut.Bordatrice.Ax.EnableStopInPhase := #MachineInterface.AckStopInPhase;
   #COut.Bordatrice.Ax.EnableStopProgrammed := #MachineInterface.AckStopProgrammed;
END_REGION

REGION Network 29: [Ax] Bordatrice - RIFERIMENTI
   RUNG wire#powerrail
      Contact( #Sts.SemiAut.ON )
      I_Contact( #AreaInterface.Cycle )
      Move(in := "A0302_Bordatrice_PERS".Par.Ax_Aut.SemiAut_Vel, out1 => #COut.Bordatrice.Ax.Vel)
      wire#w1
      Move(in := "A0302_Bordatrice_PERS".Par.Ax_Aut.Aut_Acc, out1 => #COut.Bordatrice.Ax.Acc)
      Move(in := "A0302_Bordatrice_PERS".Par.Ax_Aut.Aut_Dec, out1 => #COut.Bordatrice.Ax.Dec)
   END_RUNG
   RUNG wire#powerrail
      I_Contact( #Sts.SemiAut.ON )
      Contact( #AreaInterface.Cycle )
      Move(in := "A0302_Bordatrice_PERS".Par.Ax_Aut.Aut_Vel, out1 => #COut.Bordatrice.Ax.Vel)
   END_RUNG wire#w1
   // the same network as SCL:
   #_w1 := #Sts.SemiAut.ON AND NOT #AreaInterface.Cycle;
   IF #_w1 THEN #COut.Bordatrice.Ax.Vel := "A0302_Bordatrice_PERS".Par.Ax_Aut.SemiAut_Vel; END_IF;
   #_w2 := NOT #Sts.SemiAut.ON AND #AreaInterface.Cycle;
   IF #_w2 THEN #COut.Bordatrice.Ax.Vel := "A0302_Bordatrice_PERS".Par.Ax_Aut.Aut_Vel; END_IF;
   IF #_w1 OR #_w2 THEN
       #COut.Bordatrice.Ax.Acc := "A0302_Bordatrice_PERS".Par.Ax_Aut.Aut_Acc;
       #COut.Bordatrice.Ax.Dec := "A0302_Bordatrice_PERS".Par.Ax_Aut.Aut_Dec;
   END_IF;
END_REGION

REGION Network 31: <<<< RULLIERA >>>>
END_REGION

REGION Network 32: Rulliera - Move BTrk da Uscita Bord. Pareggiatore Coda Basso =a=> Uscita Bord. Pareggiatore Coda Alto
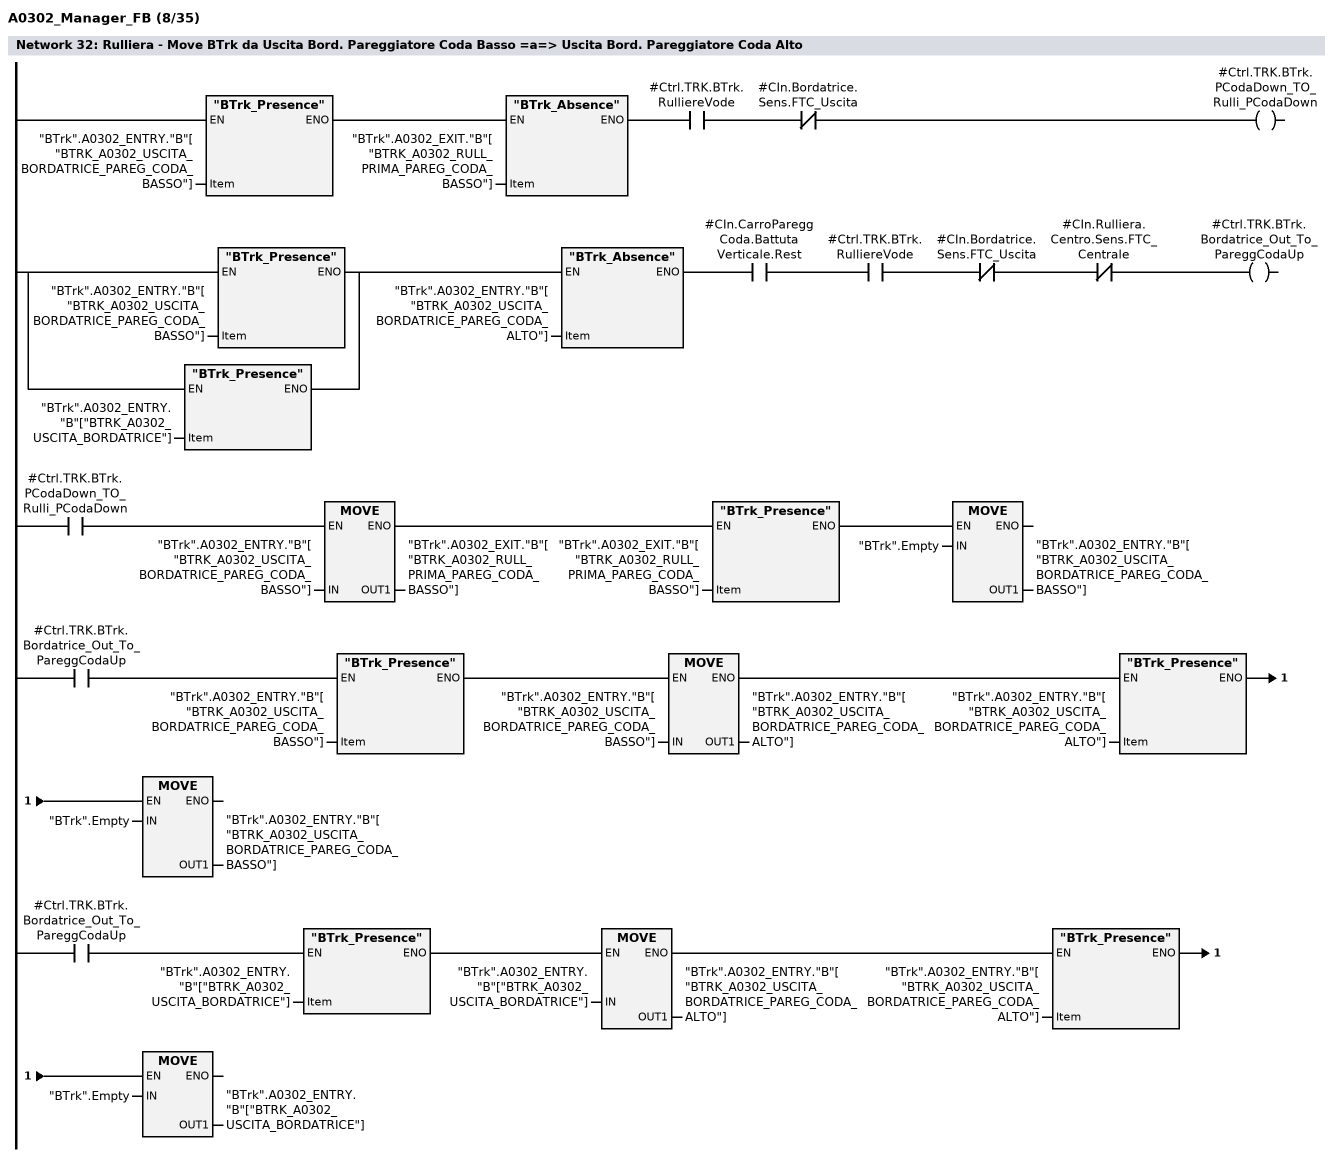
   RUNG wire#powerrail
      "BTrk_Presence"(Item := "BTrk".A0302_ENTRY."B"["BTRK_A0302_USCITA_BORDATRICE_PAREG_CODA_BASSO"])
      "BTrk_Absence"(Item := "BTrk".A0302_EXIT."B"["BTRK_A0302_RULL_PRIMA_PAREG_CODA_BASSO"])
      Contact( #Ctrl.TRK.BTrk.RulliereVode )
      I_Contact( #CIn.Bordatrice.Sens.FTC_Uscita )
      Coil( #Ctrl.TRK.BTrk.PCodaDown_TO_Rulli_PCodaDown )
   END_RUNG
   RUNG wire#powerrail
      "BTrk_Presence"(Item := "BTrk".A0302_ENTRY."B"["BTRK_A0302_USCITA_BORDATRICE_PAREG_CODA_BASSO"])
      wire#w1
      "BTrk_Absence"(Item := "BTrk".A0302_ENTRY."B"["BTRK_A0302_USCITA_BORDATRICE_PAREG_CODA_ALTO"])
      Contact( #CIn.CarroPareggCoda.BattutaVerticale.Rest )
      Contact( #Ctrl.TRK.BTrk.RulliereVode )
      I_Contact( #CIn.Bordatrice.Sens.FTC_Uscita )
      I_Contact( #CIn.Rulliera.Centro.Sens.FTC_Centrale )
      Coil( #Ctrl.TRK.BTrk.Bordatrice_Out_To_PareggCodaUp )
   END_RUNG
   RUNG wire#powerrail
      "BTrk_Presence"(Item := "BTrk".A0302_ENTRY."B"["BTRK_A0302_USCITA_BORDATRICE"])
   END_RUNG wire#w1
   RUNG wire#powerrail
      Contact( #Ctrl.TRK.BTrk.PCodaDown_TO_Rulli_PCodaDown )
      Move(in := "BTrk".A0302_ENTRY."B"["BTRK_A0302_USCITA_BORDATRICE_PAREG_CODA_BASSO"], out1 => "BTrk".A0302_EXIT."B"["BTRK_A0302_RULL_PRIMA_PAREG_CODA_BASSO"])
      "BTrk_Presence"(Item := "BTrk".A0302_EXIT."B"["BTRK_A0302_RULL_PRIMA_PAREG_CODA_BASSO"])
      Move(in := "BTrk".Empty, out1 => "BTrk".A0302_ENTRY."B"["BTRK_A0302_USCITA_BORDATRICE_PAREG_CODA_BASSO"])
   END_RUNG
   RUNG wire#powerrail
      Contact( #Ctrl.TRK.BTrk.Bordatrice_Out_To_PareggCodaUp )
      "BTrk_Presence"(Item := "BTrk".A0302_ENTRY."B"["BTRK_A0302_USCITA_BORDATRICE_PAREG_CODA_BASSO"])
      Move(in := "BTrk".A0302_ENTRY."B"["BTRK_A0302_USCITA_BORDATRICE_PAREG_CODA_BASSO"], out1 => "BTrk".A0302_ENTRY."B"["BTRK_A0302_USCITA_BORDATRICE_PAREG_CODA_ALTO"])
      "BTrk_Presence"(Item := "BTrk".A0302_ENTRY."B"["BTRK_A0302_USCITA_BORDATRICE_PAREG_CODA_ALTO"])
      Move(in := "BTrk".Empty, out1 => "BTrk".A0302_ENTRY."B"["BTRK_A0302_USCITA_BORDATRICE_PAREG_CODA_BASSO"])
   END_RUNG
   RUNG wire#powerrail
      Contact( #Ctrl.TRK.BTrk.Bordatrice_Out_To_PareggCodaUp )
      "BTrk_Presence"(Item := "BTrk".A0302_ENTRY."B"["BTRK_A0302_USCITA_BORDATRICE"])
      Move(in := "BTrk".A0302_ENTRY."B"["BTRK_A0302_USCITA_BORDATRICE"], out1 => "BTrk".A0302_ENTRY."B"["BTRK_A0302_USCITA_BORDATRICE_PAREG_CODA_ALTO"])
      "BTrk_Presence"(Item := "BTrk".A0302_ENTRY."B"["BTRK_A0302_USCITA_BORDATRICE_PAREG_CODA_ALTO"])
      Move(in := "BTrk".Empty, out1 => "BTrk".A0302_ENTRY."B"["BTRK_A0302_USCITA_BORDATRICE"])
   END_RUNG
   // the same network as SCL:
   "BTrk_Presence"(Item := "BTrk".A0302_ENTRY."B"["BTRK_A0302_USCITA_BORDATRICE_PAREG_CODA_BASSO"], ENO => #_w1);
   "BTrk_Absence"(EN := #_w1,
                  Item := "BTrk".A0302_EXIT."B"["BTRK_A0302_RULL_PRIMA_PAREG_CODA_BASSO"],
                  ENO => #_w2);
   #Ctrl.TRK.BTrk.PCodaDown_TO_Rulli_PCodaDown := #_w2 AND #Ctrl.TRK.BTrk.RulliereVode AND NOT #CIn.Bordatrice.Sens.FTC_Uscita;
   "BTrk_Presence"(Item := "BTrk".A0302_ENTRY."B"["BTRK_A0302_USCITA_BORDATRICE_PAREG_CODA_BASSO"], ENO => #_w3);
   "BTrk_Presence"(Item := "BTrk".A0302_ENTRY."B"["BTRK_A0302_USCITA_BORDATRICE"], ENO => #_w4);
   "BTrk_Absence"(EN := #_w3 OR #_w4,
                  Item := "BTrk".A0302_ENTRY."B"["BTRK_A0302_USCITA_BORDATRICE_PAREG_CODA_ALTO"],
                  ENO => #_w5);
   #Ctrl.TRK.BTrk.Bordatrice_Out_To_PareggCodaUp := #_w5 AND #CIn.CarroPareggCoda.BattutaVerticale.Rest AND #Ctrl.TRK.BTrk.RulliereVode AND NOT #CIn.Bordatrice.Sens.FTC_Uscita AND NOT #CIn.Rulliera.Centro.Sens.FTC_Centrale;
   IF #Ctrl.TRK.BTrk.PCodaDown_TO_Rulli_PCodaDown THEN
       "BTrk".A0302_EXIT."B"["BTRK_A0302_RULL_PRIMA_PAREG_CODA_BASSO"] := "BTrk".A0302_ENTRY."B"["BTRK_A0302_USCITA_BORDATRICE_PAREG_CODA_BASSO"];
   END_IF;
   "BTrk_Presence"(EN := #Ctrl.TRK.BTrk.PCodaDown_TO_Rulli_PCodaDown,
                   Item := "BTrk".A0302_EXIT."B"["BTRK_A0302_RULL_PRIMA_PAREG_CODA_BASSO"],
                   ENO => #_w6);
   IF #_w6 THEN
       "BTrk".A0302_ENTRY."B"["BTRK_A0302_USCITA_BORDATRICE_PAREG_CODA_BASSO"] := "BTrk".Empty;
   END_IF;
   "BTrk_Presence"(EN := #Ctrl.TRK.BTrk.Bordatrice_Out_To_PareggCodaUp,
                   Item := "BTrk".A0302_ENTRY."B"["BTRK_A0302_USCITA_BORDATRICE_PAREG_CODA_BASSO"],
                   ENO => #_w7);
   IF #_w7 THEN
       "BTrk".A0302_ENTRY."B"["BTRK_A0302_USCITA_BORDATRICE_PAREG_CODA_ALTO"] := "BTrk".A0302_ENTRY."B"["BTRK_A0302_USCITA_BORDATRICE_PAREG_CODA_BASSO"];
   END_IF;
   "BTrk_Presence"(EN := #_w7,
                   Item := "BTrk".A0302_ENTRY."B"["BTRK_A0302_USCITA_BORDATRICE_PAREG_CODA_ALTO"],
                   ENO => #_w8);
   IF #_w8 THEN
       "BTrk".A0302_ENTRY."B"["BTRK_A0302_USCITA_BORDATRICE_PAREG_CODA_BASSO"] := "BTrk".Empty;
   END_IF;
   "BTrk_Presence"(EN := #Ctrl.TRK.BTrk.Bordatrice_Out_To_PareggCodaUp,
                   Item := "BTrk".A0302_ENTRY."B"["BTRK_A0302_USCITA_BORDATRICE"],
                   ENO => #_w9);
   IF #_w9 THEN
       "BTrk".A0302_ENTRY."B"["BTRK_A0302_USCITA_BORDATRICE_PAREG_CODA_ALTO"] := "BTrk".A0302_ENTRY."B"["BTRK_A0302_USCITA_BORDATRICE"];
   END_IF;
   "BTrk_Presence"(EN := #_w9,
                   Item := "BTrk".A0302_ENTRY."B"["BTRK_A0302_USCITA_BORDATRICE_PAREG_CODA_ALTO"],
                   ENO => #_w10);
   IF #_w10 THEN "BTrk".A0302_ENTRY."B"["BTRK_A0302_USCITA_BORDATRICE"] := "BTrk".Empty; END_IF;
END_REGION

REGION Network 33: Rulliera - Movimento BTrk da Bordatrice-Paregg Rulliera Prima Paregg Basso => Rallenta Rulliera
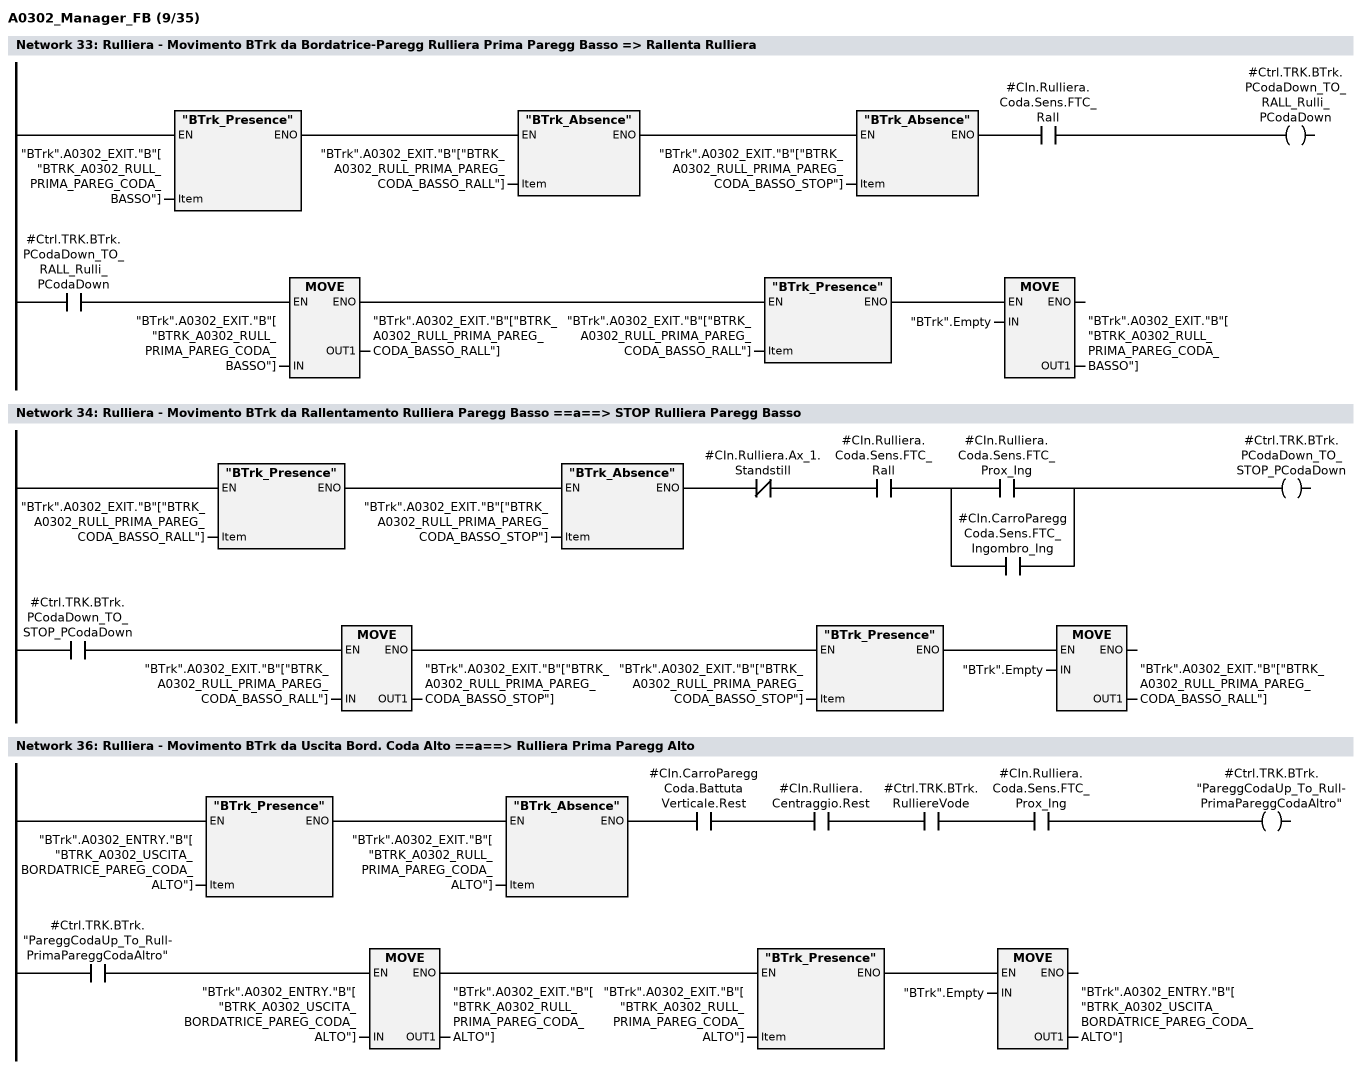
   RUNG wire#powerrail
      "BTrk_Presence"(Item := "BTrk".A0302_EXIT."B"["BTRK_A0302_RULL_PRIMA_PAREG_CODA_BASSO"])
      "BTrk_Absence"(Item := "BTrk".A0302_EXIT."B"["BTRK_A0302_RULL_PRIMA_PAREG_CODA_BASSO_RALL"])
      "BTrk_Absence"(Item := "BTrk".A0302_EXIT."B"["BTRK_A0302_RULL_PRIMA_PAREG_CODA_BASSO_STOP"])
      Contact( #CIn.Rulliera.Coda.Sens.FTC_Rall )
      Coil( #Ctrl.TRK.BTrk.PCodaDown_TO_RALL_Rulli_PCodaDown )
   END_RUNG
   RUNG wire#powerrail
      Contact( #Ctrl.TRK.BTrk.PCodaDown_TO_RALL_Rulli_PCodaDown )
      Move(in := "BTrk".A0302_EXIT."B"["BTRK_A0302_RULL_PRIMA_PAREG_CODA_BASSO"], out1 => "BTrk".A0302_EXIT."B"["BTRK_A0302_RULL_PRIMA_PAREG_CODA_BASSO_RALL"])
      "BTrk_Presence"(Item := "BTrk".A0302_EXIT."B"["BTRK_A0302_RULL_PRIMA_PAREG_CODA_BASSO_RALL"])
      Move(in := "BTrk".Empty, out1 => "BTrk".A0302_EXIT."B"["BTRK_A0302_RULL_PRIMA_PAREG_CODA_BASSO"])
   END_RUNG
   // the same network as SCL:
   "BTrk_Presence"(Item := "BTrk".A0302_EXIT."B"["BTRK_A0302_RULL_PRIMA_PAREG_CODA_BASSO"], ENO => #_w1);
   "BTrk_Absence"(EN := #_w1,
                  Item := "BTrk".A0302_EXIT."B"["BTRK_A0302_RULL_PRIMA_PAREG_CODA_BASSO_RALL"],
                  ENO => #_w2);
   "BTrk_Absence"(EN := #_w2,
                  Item := "BTrk".A0302_EXIT."B"["BTRK_A0302_RULL_PRIMA_PAREG_CODA_BASSO_STOP"],
                  ENO => #_w3);
   #Ctrl.TRK.BTrk.PCodaDown_TO_RALL_Rulli_PCodaDown := #_w3 AND #CIn.Rulliera.Coda.Sens.FTC_Rall;
   IF #Ctrl.TRK.BTrk.PCodaDown_TO_RALL_Rulli_PCodaDown THEN
       "BTrk".A0302_EXIT."B"["BTRK_A0302_RULL_PRIMA_PAREG_CODA_BASSO_RALL"] := "BTrk".A0302_EXIT."B"["BTRK_A0302_RULL_PRIMA_PAREG_CODA_BASSO"];
   END_IF;
   "BTrk_Presence"(EN := #Ctrl.TRK.BTrk.PCodaDown_TO_RALL_Rulli_PCodaDown,
                   Item := "BTrk".A0302_EXIT."B"["BTRK_A0302_RULL_PRIMA_PAREG_CODA_BASSO_RALL"],
                   ENO => #_w4);
   IF #_w4 THEN "BTrk".A0302_EXIT."B"["BTRK_A0302_RULL_PRIMA_PAREG_CODA_BASSO"] := "BTrk".Empty; END_IF;
END_REGION

REGION Network 34: Rulliera - Movimento BTrk da Rallentamento Rulliera Paregg Basso ==a==> STOP Rulliera Paregg Basso
   RUNG wire#powerrail
      "BTrk_Presence"(Item := "BTrk".A0302_EXIT."B"["BTRK_A0302_RULL_PRIMA_PAREG_CODA_BASSO_RALL"])
      "BTrk_Absence"(Item := "BTrk".A0302_EXIT."B"["BTRK_A0302_RULL_PRIMA_PAREG_CODA_BASSO_STOP"])
      I_Contact( #CIn.Rulliera.Ax_1.Standstill )
      Contact( #CIn.Rulliera.Coda.Sens.FTC_Rall )
      wire#w1
      Contact( #CIn.Rulliera.Coda.Sens.FTC_Prox_Ing )
      wire#w2
      Coil( #Ctrl.TRK.BTrk.PCodaDown_TO_STOP_PCodaDown )
   END_RUNG
   RUNG wire#w1
      Contact( #CIn.CarroPareggCoda.Sens.FTC_Ingombro_Ing )
   END_RUNG wire#w2
   RUNG wire#powerrail
      Contact( #Ctrl.TRK.BTrk.PCodaDown_TO_STOP_PCodaDown )
      Move(in := "BTrk".A0302_EXIT."B"["BTRK_A0302_RULL_PRIMA_PAREG_CODA_BASSO_RALL"], out1 => "BTrk".A0302_EXIT."B"["BTRK_A0302_RULL_PRIMA_PAREG_CODA_BASSO_STOP"])
      "BTrk_Presence"(Item := "BTrk".A0302_EXIT."B"["BTRK_A0302_RULL_PRIMA_PAREG_CODA_BASSO_STOP"])
      Move(in := "BTrk".Empty, out1 => "BTrk".A0302_EXIT."B"["BTRK_A0302_RULL_PRIMA_PAREG_CODA_BASSO_RALL"])
   END_RUNG
   // the same network as SCL:
   "BTrk_Presence"(Item := "BTrk".A0302_EXIT."B"["BTRK_A0302_RULL_PRIMA_PAREG_CODA_BASSO_RALL"], ENO => #_w1);
   "BTrk_Absence"(EN := #_w1,
                  Item := "BTrk".A0302_EXIT."B"["BTRK_A0302_RULL_PRIMA_PAREG_CODA_BASSO_STOP"],
                  ENO => #_w2);
   #Ctrl.TRK.BTrk.PCodaDown_TO_STOP_PCodaDown := #_w2 AND NOT #CIn.Rulliera.Ax_1.Standstill AND #CIn.Rulliera.Coda.Sens.FTC_Rall AND (#CIn.Rulliera.Coda.Sens.FTC_Prox_Ing OR #CIn.CarroPareggCoda.Sens.FTC_Ingombro_Ing);
   IF #Ctrl.TRK.BTrk.PCodaDown_TO_STOP_PCodaDown THEN
       "BTrk".A0302_EXIT."B"["BTRK_A0302_RULL_PRIMA_PAREG_CODA_BASSO_STOP"] := "BTrk".A0302_EXIT."B"["BTRK_A0302_RULL_PRIMA_PAREG_CODA_BASSO_RALL"];
   END_IF;
   "BTrk_Presence"(EN := #Ctrl.TRK.BTrk.PCodaDown_TO_STOP_PCodaDown,
                   Item := "BTrk".A0302_EXIT."B"["BTRK_A0302_RULL_PRIMA_PAREG_CODA_BASSO_STOP"],
                   ENO => #_w3);
   IF #_w3 THEN "BTrk".A0302_EXIT."B"["BTRK_A0302_RULL_PRIMA_PAREG_CODA_BASSO_RALL"] := "BTrk".Empty; END_IF;
END_REGION

REGION Network 36: Rulliera - Movimento BTrk da Uscita Bord. Coda Alto ==a==> Rulliera Prima Paregg Alto
   RUNG wire#powerrail
      "BTrk_Presence"(Item := "BTrk".A0302_ENTRY."B"["BTRK_A0302_USCITA_BORDATRICE_PAREG_CODA_ALTO"])
      "BTrk_Absence"(Item := "BTrk".A0302_EXIT."B"["BTRK_A0302_RULL_PRIMA_PAREG_CODA_ALTO"])
      Contact( #CIn.CarroPareggCoda.BattutaVerticale.Rest )
      Contact( #CIn.Rulliera.Centraggio.Rest )
      Contact( #Ctrl.TRK.BTrk.RulliereVode )
      Contact( #CIn.Rulliera.Coda.Sens.FTC_Prox_Ing )
      Coil( #Ctrl.TRK.BTrk."PareggCodaUp_To_Rull-PrimaPareggCodaAltro" )
   END_RUNG
   RUNG wire#powerrail
      Contact( #Ctrl.TRK.BTrk."PareggCodaUp_To_Rull-PrimaPareggCodaAltro" )
      Move(in := "BTrk".A0302_ENTRY."B"["BTRK_A0302_USCITA_BORDATRICE_PAREG_CODA_ALTO"], out1 => "BTrk".A0302_EXIT."B"["BTRK_A0302_RULL_PRIMA_PAREG_CODA_ALTO"])
      "BTrk_Presence"(Item := "BTrk".A0302_EXIT."B"["BTRK_A0302_RULL_PRIMA_PAREG_CODA_ALTO"])
      Move(in := "BTrk".Empty, out1 => "BTrk".A0302_ENTRY."B"["BTRK_A0302_USCITA_BORDATRICE_PAREG_CODA_ALTO"])
   END_RUNG
   // the same network as SCL:
   "BTrk_Presence"(Item := "BTrk".A0302_ENTRY."B"["BTRK_A0302_USCITA_BORDATRICE_PAREG_CODA_ALTO"], ENO => #_w1);
   "BTrk_Absence"(EN := #_w1,
                  Item := "BTrk".A0302_EXIT."B"["BTRK_A0302_RULL_PRIMA_PAREG_CODA_ALTO"],
                  ENO => #_w2);
   #Ctrl.TRK.BTrk."PareggCodaUp_To_Rull-PrimaPareggCodaAltro" := #_w2 AND #CIn.CarroPareggCoda.BattutaVerticale.Rest AND #CIn.Rulliera.Centraggio.Rest AND #Ctrl.TRK.BTrk.RulliereVode AND #CIn.Rulliera.Coda.Sens.FTC_Prox_Ing;
   IF #Ctrl.TRK.BTrk."PareggCodaUp_To_Rull-PrimaPareggCodaAltro" THEN
       "BTrk".A0302_EXIT."B"["BTRK_A0302_RULL_PRIMA_PAREG_CODA_ALTO"] := "BTrk".A0302_ENTRY."B"["BTRK_A0302_USCITA_BORDATRICE_PAREG_CODA_ALTO"];
   END_IF;
   "BTrk_Presence"(EN := #Ctrl.TRK.BTrk."PareggCodaUp_To_Rull-PrimaPareggCodaAltro",
                   Item := "BTrk".A0302_EXIT."B"["BTRK_A0302_RULL_PRIMA_PAREG_CODA_ALTO"],
                   ENO => #_w3);
   IF #_w3 THEN
       "BTrk".A0302_ENTRY."B"["BTRK_A0302_USCITA_BORDATRICE_PAREG_CODA_ALTO"] := "BTrk".Empty;
   END_IF;
END_REGION

REGION Network 37: <+>
END_REGION

REGION Network 38: ########### [Ax] Rulliera - Controllo condizioni di START - Fwd ################
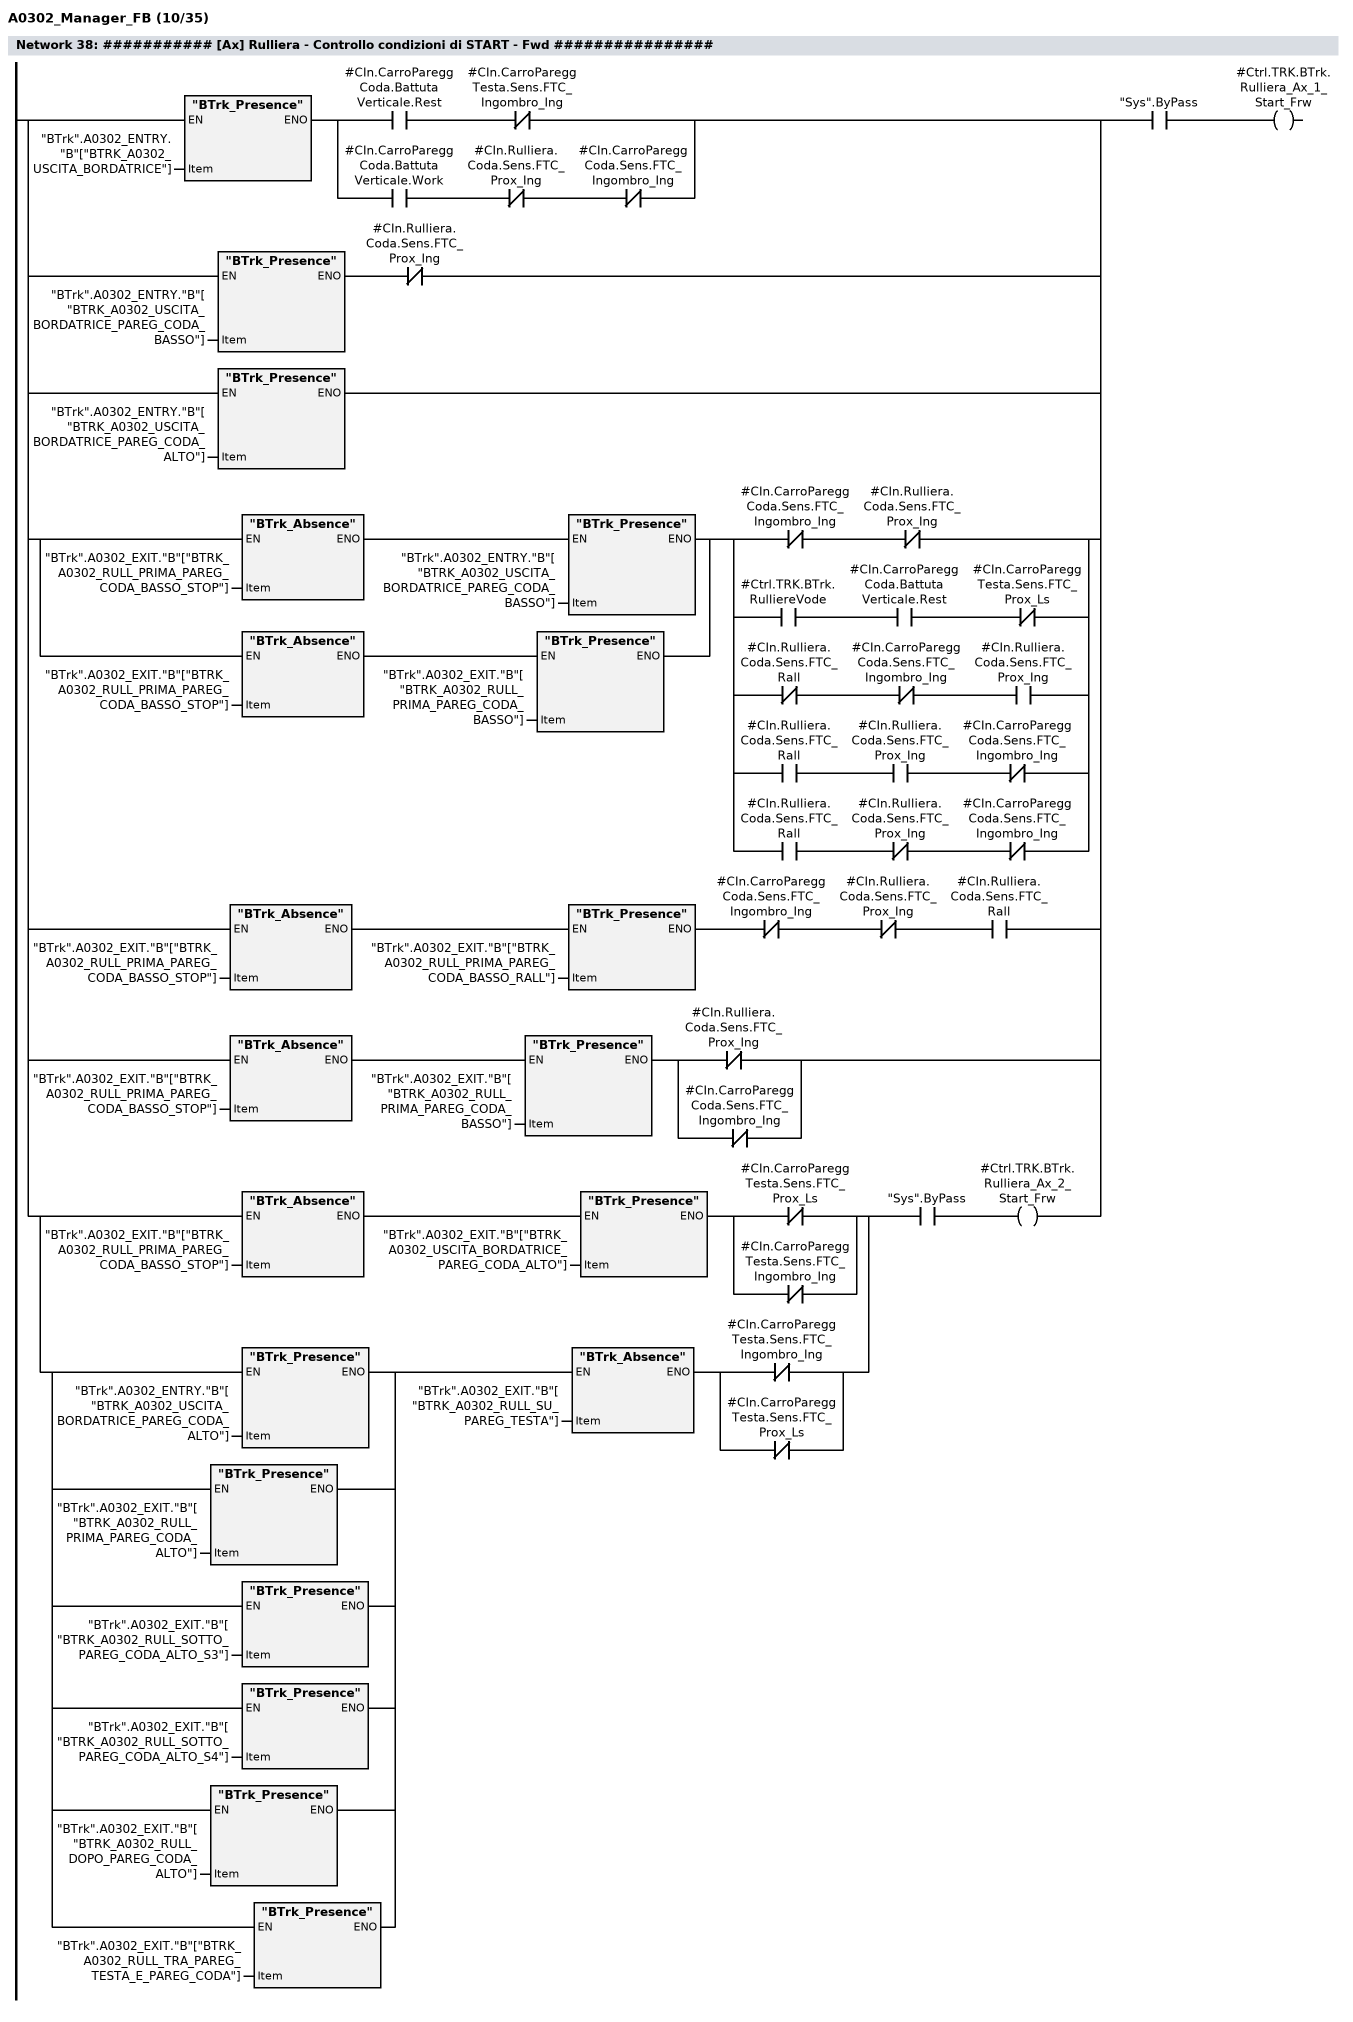
   RUNG wire#powerrail
      "BTrk_Presence"(Item := "BTrk".A0302_ENTRY."B"["BTRK_A0302_USCITA_BORDATRICE"])
      wire#w1
      Contact( #CIn.CarroPareggCoda.BattutaVerticale.Rest )
      I_Contact( #CIn.CarroPareggTesta.Sens.FTC_Ingombro_Ing )
      wire#w2
      Contact( "Sys".ByPass )
      Coil( #Ctrl.TRK.BTrk.Rulliera_Ax_1_Start_Frw )
   END_RUNG
   RUNG wire#w1
      Contact( #CIn.CarroPareggCoda.BattutaVerticale.Work )
      I_Contact( #CIn.Rulliera.Coda.Sens.FTC_Prox_Ing )
      I_Contact( #CIn.CarroPareggCoda.Sens.FTC_Ingombro_Ing )
   END_RUNG wire#w2
   RUNG wire#powerrail
      "BTrk_Presence"(Item := "BTrk".A0302_ENTRY."B"["BTRK_A0302_USCITA_BORDATRICE_PAREG_CODA_BASSO"])
      I_Contact( #CIn.Rulliera.Coda.Sens.FTC_Prox_Ing )
   END_RUNG wire#w2
   RUNG wire#powerrail
      "BTrk_Presence"(Item := "BTrk".A0302_ENTRY."B"["BTRK_A0302_USCITA_BORDATRICE_PAREG_CODA_ALTO"])
   END_RUNG wire#w2
   RUNG wire#powerrail
      "BTrk_Absence"(Item := "BTrk".A0302_EXIT."B"["BTRK_A0302_RULL_PRIMA_PAREG_CODA_BASSO_STOP"])
      "BTrk_Presence"(Item := "BTrk".A0302_ENTRY."B"["BTRK_A0302_USCITA_BORDATRICE_PAREG_CODA_BASSO"])
      wire#w3
      I_Contact( #CIn.CarroPareggCoda.Sens.FTC_Ingombro_Ing )
      I_Contact( #CIn.Rulliera.Coda.Sens.FTC_Prox_Ing )
   END_RUNG wire#w2
   RUNG wire#powerrail
      "BTrk_Absence"(Item := "BTrk".A0302_EXIT."B"["BTRK_A0302_RULL_PRIMA_PAREG_CODA_BASSO_STOP"])
      "BTrk_Presence"(Item := "BTrk".A0302_EXIT."B"["BTRK_A0302_RULL_PRIMA_PAREG_CODA_BASSO"])
   END_RUNG wire#w3
   RUNG wire#w3
      Contact( #Ctrl.TRK.BTrk.RulliereVode )
      Contact( #CIn.CarroPareggCoda.BattutaVerticale.Rest )
      I_Contact( #CIn.CarroPareggTesta.Sens.FTC_Prox_Ls )
   END_RUNG wire#w2
   RUNG wire#w3
      I_Contact( #CIn.Rulliera.Coda.Sens.FTC_Rall )
      I_Contact( #CIn.CarroPareggCoda.Sens.FTC_Ingombro_Ing )
      Contact( #CIn.Rulliera.Coda.Sens.FTC_Prox_Ing )
   END_RUNG wire#w2
   RUNG wire#w3
      Contact( #CIn.Rulliera.Coda.Sens.FTC_Rall )
      Contact( #CIn.Rulliera.Coda.Sens.FTC_Prox_Ing )
      I_Contact( #CIn.CarroPareggCoda.Sens.FTC_Ingombro_Ing )
   END_RUNG wire#w2
   RUNG wire#w3
      Contact( #CIn.Rulliera.Coda.Sens.FTC_Rall )
      I_Contact( #CIn.Rulliera.Coda.Sens.FTC_Prox_Ing )
      I_Contact( #CIn.CarroPareggCoda.Sens.FTC_Ingombro_Ing )
   END_RUNG wire#w2
   RUNG wire#powerrail
      "BTrk_Absence"(Item := "BTrk".A0302_EXIT."B"["BTRK_A0302_RULL_PRIMA_PAREG_CODA_BASSO_STOP"])
      "BTrk_Presence"(Item := "BTrk".A0302_EXIT."B"["BTRK_A0302_RULL_PRIMA_PAREG_CODA_BASSO_RALL"])
      I_Contact( #CIn.CarroPareggCoda.Sens.FTC_Ingombro_Ing )
      I_Contact( #CIn.Rulliera.Coda.Sens.FTC_Prox_Ing )
      Contact( #CIn.Rulliera.Coda.Sens.FTC_Rall )
   END_RUNG wire#w2
   RUNG wire#powerrail
      "BTrk_Absence"(Item := "BTrk".A0302_EXIT."B"["BTRK_A0302_RULL_PRIMA_PAREG_CODA_BASSO_STOP"])
      "BTrk_Presence"(Item := "BTrk".A0302_EXIT."B"["BTRK_A0302_RULL_PRIMA_PAREG_CODA_BASSO"])
      wire#w4
      I_Contact( #CIn.Rulliera.Coda.Sens.FTC_Prox_Ing )
   END_RUNG wire#w2
   RUNG wire#w4
      I_Contact( #CIn.CarroPareggCoda.Sens.FTC_Ingombro_Ing )
   END_RUNG wire#w2
   RUNG wire#powerrail
      "BTrk_Absence"(Item := "BTrk".A0302_EXIT."B"["BTRK_A0302_RULL_PRIMA_PAREG_CODA_BASSO_STOP"])
      "BTrk_Presence"(Item := "BTrk".A0302_EXIT."B"["BTRK_A0302_USCITA_BORDATRICE_PAREG_CODA_ALTO"])
      wire#w5
      I_Contact( #CIn.CarroPareggTesta.Sens.FTC_Prox_Ls )
      wire#w6
      Contact( "Sys".ByPass )
      Coil( #Ctrl.TRK.BTrk.Rulliera_Ax_2_Start_Frw )
   END_RUNG wire#w2
   RUNG wire#w5
      I_Contact( #CIn.CarroPareggTesta.Sens.FTC_Ingombro_Ing )
   END_RUNG wire#w6
   RUNG wire#powerrail
      "BTrk_Presence"(Item := "BTrk".A0302_ENTRY."B"["BTRK_A0302_USCITA_BORDATRICE_PAREG_CODA_ALTO"])
      wire#w7
      "BTrk_Absence"(Item := "BTrk".A0302_EXIT."B"["BTRK_A0302_RULL_SU_PAREG_TESTA"])
      wire#w8
      I_Contact( #CIn.CarroPareggTesta.Sens.FTC_Ingombro_Ing )
   END_RUNG wire#w6
   RUNG wire#powerrail
      "BTrk_Presence"(Item := "BTrk".A0302_EXIT."B"["BTRK_A0302_RULL_PRIMA_PAREG_CODA_ALTO"])
   END_RUNG wire#w7
   RUNG wire#powerrail
      "BTrk_Presence"(Item := "BTrk".A0302_EXIT."B"["BTRK_A0302_RULL_SOTTO_PAREG_CODA_ALTO_S3"])
   END_RUNG wire#w7
   RUNG wire#powerrail
      "BTrk_Presence"(Item := "BTrk".A0302_EXIT."B"["BTRK_A0302_RULL_SOTTO_PAREG_CODA_ALTO_S4"])
   END_RUNG wire#w7
   RUNG wire#powerrail
      "BTrk_Presence"(Item := "BTrk".A0302_EXIT."B"["BTRK_A0302_RULL_DOPO_PAREG_CODA_ALTO"])
   END_RUNG wire#w7
   RUNG wire#powerrail
      "BTrk_Presence"(Item := "BTrk".A0302_EXIT."B"["BTRK_A0302_RULL_TRA_PAREG_TESTA_E_PAREG_CODA"])
   END_RUNG wire#w7
   RUNG wire#w8
      I_Contact( #CIn.CarroPareggTesta.Sens.FTC_Prox_Ls )
   END_RUNG wire#w6
   // the same network as SCL:
   "BTrk_Presence"(Item := "BTrk".A0302_ENTRY."B"["BTRK_A0302_USCITA_BORDATRICE"], ENO => #_w1);
   "BTrk_Presence"(Item := "BTrk".A0302_ENTRY."B"["BTRK_A0302_USCITA_BORDATRICE_PAREG_CODA_BASSO"], ENO => #_w2);
   "BTrk_Presence"(Item := "BTrk".A0302_ENTRY."B"["BTRK_A0302_USCITA_BORDATRICE_PAREG_CODA_ALTO"], ENO => #_w3);
   "BTrk_Absence"(Item := "BTrk".A0302_EXIT."B"["BTRK_A0302_RULL_PRIMA_PAREG_CODA_BASSO_STOP"], ENO => #_w4);
   "BTrk_Presence"(EN := #_w4,
                   Item := "BTrk".A0302_ENTRY."B"["BTRK_A0302_USCITA_BORDATRICE_PAREG_CODA_BASSO"],
                   ENO => #_w5);
   "BTrk_Absence"(Item := "BTrk".A0302_EXIT."B"["BTRK_A0302_RULL_PRIMA_PAREG_CODA_BASSO_STOP"], ENO => #_w6);
   "BTrk_Presence"(EN := #_w6,
                   Item := "BTrk".A0302_EXIT."B"["BTRK_A0302_RULL_PRIMA_PAREG_CODA_BASSO"],
                   ENO => #_w7);
   "BTrk_Absence"(Item := "BTrk".A0302_EXIT."B"["BTRK_A0302_RULL_PRIMA_PAREG_CODA_BASSO_STOP"], ENO => #_w8);
   "BTrk_Presence"(EN := #_w8,
                   Item := "BTrk".A0302_EXIT."B"["BTRK_A0302_RULL_PRIMA_PAREG_CODA_BASSO_RALL"],
                   ENO => #_w9);
   "BTrk_Absence"(Item := "BTrk".A0302_EXIT."B"["BTRK_A0302_RULL_PRIMA_PAREG_CODA_BASSO_STOP"], ENO => #_w10);
   "BTrk_Presence"(EN := #_w10,
                   Item := "BTrk".A0302_EXIT."B"["BTRK_A0302_RULL_PRIMA_PAREG_CODA_BASSO"],
                   ENO => #_w11);
   "BTrk_Absence"(Item := "BTrk".A0302_EXIT."B"["BTRK_A0302_RULL_PRIMA_PAREG_CODA_BASSO_STOP"], ENO => #_w12);
   "BTrk_Presence"(EN := #_w12,
                   Item := "BTrk".A0302_EXIT."B"["BTRK_A0302_USCITA_BORDATRICE_PAREG_CODA_ALTO"],
                   ENO => #_w13);
   "BTrk_Presence"(Item := "BTrk".A0302_ENTRY."B"["BTRK_A0302_USCITA_BORDATRICE_PAREG_CODA_ALTO"], ENO => #_w14);
   "BTrk_Presence"(Item := "BTrk".A0302_EXIT."B"["BTRK_A0302_RULL_PRIMA_PAREG_CODA_ALTO"], ENO => #_w15);
   "BTrk_Presence"(Item := "BTrk".A0302_EXIT."B"["BTRK_A0302_RULL_SOTTO_PAREG_CODA_ALTO_S3"], ENO => #_w16);
   "BTrk_Presence"(Item := "BTrk".A0302_EXIT."B"["BTRK_A0302_RULL_SOTTO_PAREG_CODA_ALTO_S4"], ENO => #_w17);
   "BTrk_Presence"(Item := "BTrk".A0302_EXIT."B"["BTRK_A0302_RULL_DOPO_PAREG_CODA_ALTO"], ENO => #_w18);
   "BTrk_Presence"(Item := "BTrk".A0302_EXIT."B"["BTRK_A0302_RULL_TRA_PAREG_TESTA_E_PAREG_CODA"], ENO => #_w19);
   "BTrk_Absence"(EN := #_w14 OR #_w15 OR #_w16 OR #_w17 OR #_w18 OR #_w19,
                  Item := "BTrk".A0302_EXIT."B"["BTRK_A0302_RULL_SU_PAREG_TESTA"],
                  ENO => #_w20);
   #Ctrl.TRK.BTrk.Rulliera_Ax_2_Start_Frw := ((#_w13 AND (NOT #CIn.CarroPareggTesta.Sens.FTC_Prox_Ls OR NOT #CIn.CarroPareggTesta.Sens.FTC_Ingombro_Ing)) OR (#_w20 AND (NOT #CIn.CarroPareggTesta.Sens.FTC_Ingombro_Ing OR NOT #CIn.CarroPareggTesta.Sens.FTC_Prox_Ls))) AND "Sys".ByPass;
   #Ctrl.TRK.BTrk.Rulliera_Ax_1_Start_Frw := ((#_w1 AND ((#CIn.CarroPareggCoda.BattutaVerticale.Rest AND NOT #CIn.CarroPareggTesta.Sens.FTC_Ingombro_Ing) OR (#CIn.CarroPareggCoda.BattutaVerticale.Work AND NOT #CIn.Rulliera.Coda.Sens.FTC_Prox_Ing AND NOT #CIn.CarroPareggCoda.Sens.FTC_Ingombro_Ing))) OR (#_w2 AND NOT #CIn.Rulliera.Coda.Sens.FTC_Prox_Ing) OR #_w3 OR ((#_w5 OR #_w7) AND ((NOT #CIn.CarroPareggCoda.Sens.FTC_Ingombro_Ing AND NOT #CIn.Rulliera.Coda.Sens.FTC_Prox_Ing) OR (#Ctrl.TRK.BTrk.RulliereVode AND #CIn.CarroPareggCoda.BattutaVerticale.Rest AND NOT #CIn.CarroPareggTesta.Sens.FTC_Prox_Ls) OR (NOT #CIn.Rulliera.Coda.Sens.FTC_Rall AND NOT #CIn.CarroPareggCoda.Sens.FTC_Ingombro_Ing AND #CIn.Rulliera.Coda.Sens.FTC_Prox_Ing) OR (#CIn.Rulliera.Coda.Sens.FTC_Rall AND #CIn.Rulliera.Coda.Sens.FTC_Prox_Ing AND NOT #CIn.CarroPareggCoda.Sens.FTC_Ingombro_Ing) OR (#CIn.Rulliera.Coda.Sens.FTC_Rall AND NOT #CIn.Rulliera.Coda.Sens.FTC_Prox_Ing AND NOT #CIn.CarroPareggCoda.Sens.FTC_Ingombro_Ing))) OR (#_w9 AND NOT #CIn.CarroPareggCoda.Sens.FTC_Ingombro_Ing AND NOT #CIn.Rulliera.Coda.Sens.FTC_Prox_Ing AND #CIn.Rulliera.Coda.Sens.FTC_Rall) OR (#_w11 AND (NOT #CIn.Rulliera.Coda.Sens.FTC_Prox_Ing OR NOT #CIn.CarroPareggCoda.Sens.FTC_Ingombro_Ing)) OR #Ctrl.TRK.BTrk.Rulliera_Ax_2_Start_Frw) AND "Sys".ByPass;
END_REGION

REGION Network 39: [Ax] Rulliera - Controllo condizioni di START - Fwd a velocità Bordatrice
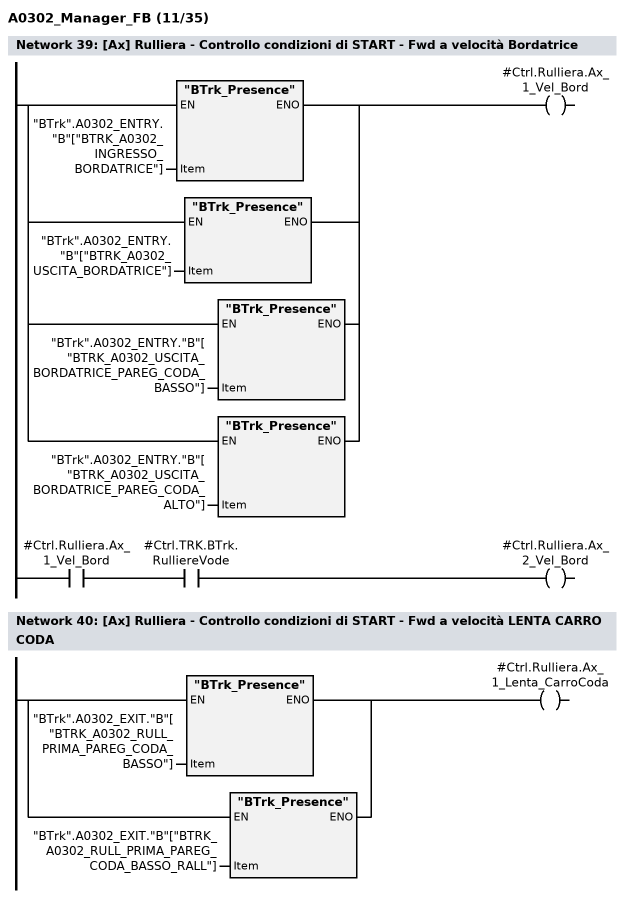
   RUNG wire#powerrail
      "BTrk_Presence"(Item := "BTrk".A0302_ENTRY."B"["BTRK_A0302_INGRESSO_BORDATRICE"])
      wire#w1
      Coil( #Ctrl.Rulliera.Ax_1_Vel_Bord )
   END_RUNG
   RUNG wire#powerrail
      "BTrk_Presence"(Item := "BTrk".A0302_ENTRY."B"["BTRK_A0302_USCITA_BORDATRICE"])
   END_RUNG wire#w1
   RUNG wire#powerrail
      "BTrk_Presence"(Item := "BTrk".A0302_ENTRY."B"["BTRK_A0302_USCITA_BORDATRICE_PAREG_CODA_BASSO"])
   END_RUNG wire#w1
   RUNG wire#powerrail
      "BTrk_Presence"(Item := "BTrk".A0302_ENTRY."B"["BTRK_A0302_USCITA_BORDATRICE_PAREG_CODA_ALTO"])
   END_RUNG wire#w1
   RUNG wire#powerrail
      Contact( #Ctrl.Rulliera.Ax_1_Vel_Bord )
      Contact( #Ctrl.TRK.BTrk.RulliereVode )
      Coil( #Ctrl.Rulliera.Ax_2_Vel_Bord )
   END_RUNG
   // the same network as SCL:
   "BTrk_Presence"(Item := "BTrk".A0302_ENTRY."B"["BTRK_A0302_INGRESSO_BORDATRICE"], ENO => #_w1);
   "BTrk_Presence"(Item := "BTrk".A0302_ENTRY."B"["BTRK_A0302_USCITA_BORDATRICE"], ENO => #_w2);
   "BTrk_Presence"(Item := "BTrk".A0302_ENTRY."B"["BTRK_A0302_USCITA_BORDATRICE_PAREG_CODA_BASSO"], ENO => #_w3);
   "BTrk_Presence"(Item := "BTrk".A0302_ENTRY."B"["BTRK_A0302_USCITA_BORDATRICE_PAREG_CODA_ALTO"], ENO => #_w4);
   #Ctrl.Rulliera.Ax_1_Vel_Bord := #_w1 OR #_w2 OR #_w3 OR #_w4;
   #Ctrl.Rulliera.Ax_2_Vel_Bord := #Ctrl.Rulliera.Ax_1_Vel_Bord AND #Ctrl.TRK.BTrk.RulliereVode;
END_REGION

REGION Network 40: [Ax] Rulliera - Controllo condizioni di START - Fwd a velocità LENTA CARRO CODA
   RUNG wire#powerrail
      "BTrk_Presence"(Item := "BTrk".A0302_EXIT."B"["BTRK_A0302_RULL_PRIMA_PAREG_CODA_BASSO"])
      wire#w1
      Coil( #Ctrl.Rulliera.Ax_1_Lenta_CarroCoda )
   END_RUNG
   RUNG wire#powerrail
      "BTrk_Presence"(Item := "BTrk".A0302_EXIT."B"["BTRK_A0302_RULL_PRIMA_PAREG_CODA_BASSO_RALL"])
   END_RUNG wire#w1
   // the same network as SCL:
   "BTrk_Presence"(Item := "BTrk".A0302_EXIT."B"["BTRK_A0302_RULL_PRIMA_PAREG_CODA_BASSO"], ENO => #_w1);
   "BTrk_Presence"(Item := "BTrk".A0302_EXIT."B"["BTRK_A0302_RULL_PRIMA_PAREG_CODA_BASSO_RALL"], ENO => #_w2);
   #Ctrl.Rulliera.Ax_1_Lenta_CarroCoda := #_w1 OR #_w2;
END_REGION

REGION Network 41: [Ax] Rulliera - Controllo condizioni di START - Fwd Velocità CARRO TESTA
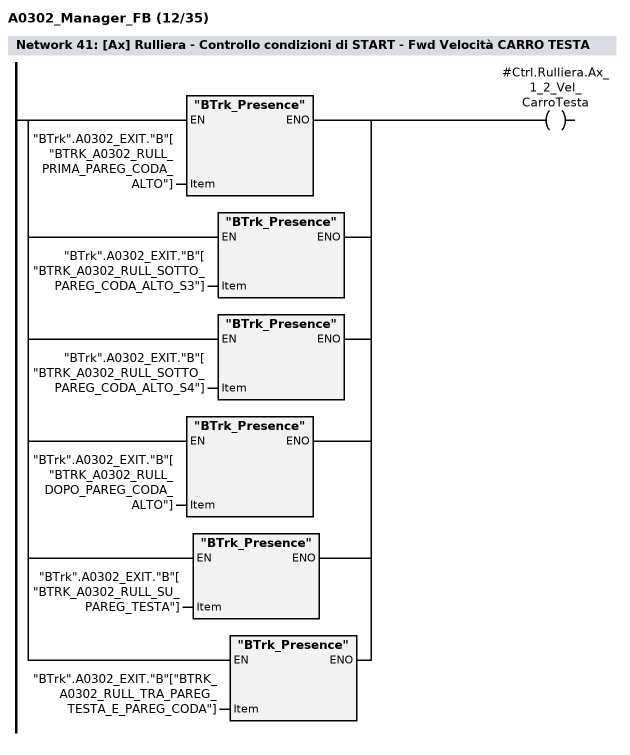
   RUNG wire#powerrail
      "BTrk_Presence"(Item := "BTrk".A0302_EXIT."B"["BTRK_A0302_RULL_PRIMA_PAREG_CODA_ALTO"])
      wire#w1
      Coil( #Ctrl.Rulliera.Ax_1_2_Vel_CarroTesta )
   END_RUNG
   RUNG wire#powerrail
      "BTrk_Presence"(Item := "BTrk".A0302_EXIT."B"["BTRK_A0302_RULL_SOTTO_PAREG_CODA_ALTO_S3"])
   END_RUNG wire#w1
   RUNG wire#powerrail
      "BTrk_Presence"(Item := "BTrk".A0302_EXIT."B"["BTRK_A0302_RULL_SOTTO_PAREG_CODA_ALTO_S4"])
   END_RUNG wire#w1
   RUNG wire#powerrail
      "BTrk_Presence"(Item := "BTrk".A0302_EXIT."B"["BTRK_A0302_RULL_DOPO_PAREG_CODA_ALTO"])
   END_RUNG wire#w1
   RUNG wire#powerrail
      "BTrk_Presence"(Item := "BTrk".A0302_EXIT."B"["BTRK_A0302_RULL_SU_PAREG_TESTA"])
   END_RUNG wire#w1
   RUNG wire#powerrail
      "BTrk_Presence"(Item := "BTrk".A0302_EXIT."B"["BTRK_A0302_RULL_TRA_PAREG_TESTA_E_PAREG_CODA"])
   END_RUNG wire#w1
   // the same network as SCL:
   "BTrk_Presence"(Item := "BTrk".A0302_EXIT."B"["BTRK_A0302_RULL_PRIMA_PAREG_CODA_ALTO"], ENO => #_w1);
   "BTrk_Presence"(Item := "BTrk".A0302_EXIT."B"["BTRK_A0302_RULL_SOTTO_PAREG_CODA_ALTO_S3"], ENO => #_w2);
   "BTrk_Presence"(Item := "BTrk".A0302_EXIT."B"["BTRK_A0302_RULL_SOTTO_PAREG_CODA_ALTO_S4"], ENO => #_w3);
   "BTrk_Presence"(Item := "BTrk".A0302_EXIT."B"["BTRK_A0302_RULL_DOPO_PAREG_CODA_ALTO"], ENO => #_w4);
   "BTrk_Presence"(Item := "BTrk".A0302_EXIT."B"["BTRK_A0302_RULL_SU_PAREG_TESTA"], ENO => #_w5);
   "BTrk_Presence"(Item := "BTrk".A0302_EXIT."B"["BTRK_A0302_RULL_TRA_PAREG_TESTA_E_PAREG_CODA"], ENO => #_w6);
   #Ctrl.Rulliera.Ax_1_2_Vel_CarroTesta := #_w1 OR #_w2 OR #_w3 OR #_w4 OR #_w5 OR #_w6;
END_REGION

REGION Network 42: [Ax] Rulliera - Rallentamento Rulliera Calcolato
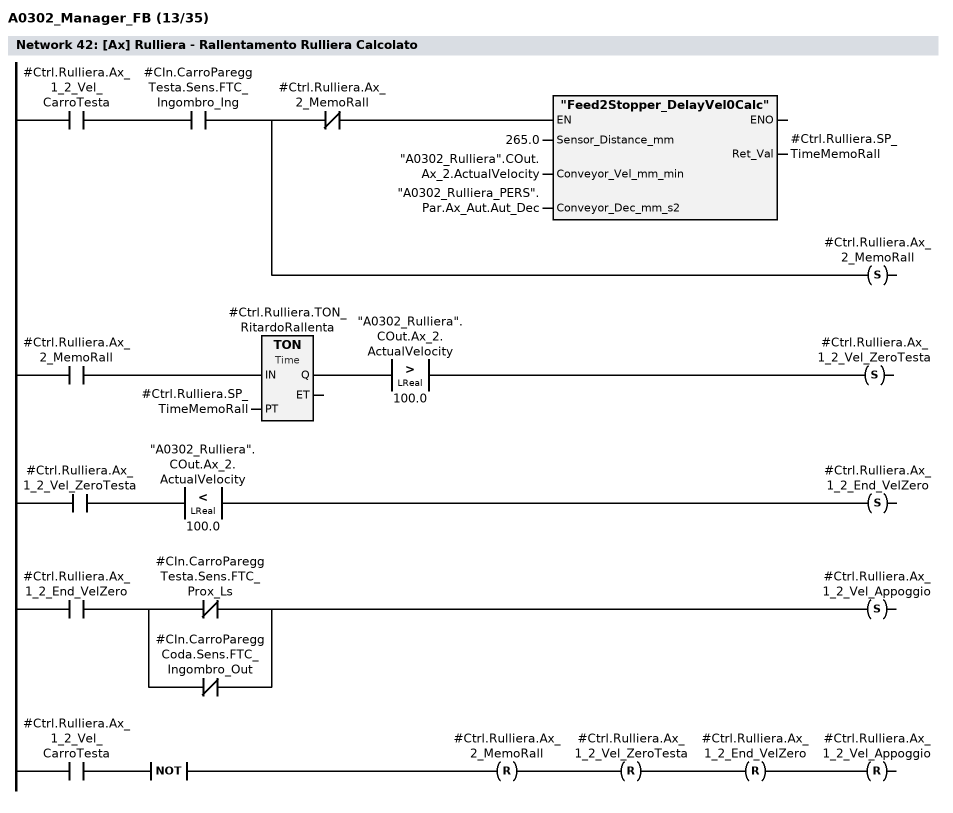
   RUNG wire#powerrail
      Contact( #Ctrl.Rulliera.Ax_1_2_Vel_CarroTesta )
      Contact( #CIn.CarroPareggTesta.Sens.FTC_Ingombro_Ing )
      wire#w1
      I_Contact( #Ctrl.Rulliera.Ax_2_MemoRall )
      "Feed2Stopper_DelayVel0Calc"(Sensor_Distance_mm := 265.0, Conveyor_Vel_mm_min := "A0302_Rulliera".COut.Ax_2.ActualVelocity, Conveyor_Dec_mm_s2 := "A0302_Rulliera_PERS".Par.Ax_Aut.Aut_Dec, Ret_Val => #Ctrl.Rulliera.SP_TimeMemoRall)
   END_RUNG
   RUNG wire#w1
      S_Coil( #Ctrl.Rulliera.Ax_2_MemoRall )
   END_RUNG
   RUNG wire#powerrail
      Contact( #Ctrl.Rulliera.Ax_2_MemoRall )
      { S7_Templates := "time_type := Time" } #Ctrl.Rulliera.TON_RitardoRallenta.TON(pt := #Ctrl.Rulliera.SP_TimeMemoRall, et =>)
      { S7_Templates := "SrcType := LReal" } GT_Contact(in1 := "A0302_Rulliera".COut.Ax_2.ActualVelocity, in2 := 100.0)
      S_Coil( #Ctrl.Rulliera.Ax_1_2_Vel_ZeroTesta )
   END_RUNG
   RUNG wire#powerrail
      Contact( #Ctrl.Rulliera.Ax_1_2_Vel_ZeroTesta )
      { S7_Templates := "SrcType := LReal" } LT_Contact(in1 := "A0302_Rulliera".COut.Ax_2.ActualVelocity, in2 := 100.0)
      S_Coil( #Ctrl.Rulliera.Ax_1_2_End_VelZero )
   END_RUNG
   RUNG wire#powerrail
      Contact( #Ctrl.Rulliera.Ax_1_2_End_VelZero )
      wire#w2
      I_Contact( #CIn.CarroPareggTesta.Sens.FTC_Prox_Ls )
      wire#w3
      S_Coil( #Ctrl.Rulliera.Ax_1_2_Vel_Appoggio )
   END_RUNG
   RUNG wire#w2
      I_Contact( #CIn.CarroPareggCoda.Sens.FTC_Ingombro_Out )
   END_RUNG wire#w3
   RUNG wire#powerrail
      Contact( #Ctrl.Rulliera.Ax_1_2_Vel_CarroTesta )
      Not()
      R_Coil( #Ctrl.Rulliera.Ax_2_MemoRall )
      R_Coil( #Ctrl.Rulliera.Ax_1_2_Vel_ZeroTesta )
      R_Coil( #Ctrl.Rulliera.Ax_1_2_End_VelZero )
      R_Coil( #Ctrl.Rulliera.Ax_1_2_Vel_Appoggio )
   END_RUNG
   // the same network as SCL:
   #_w1 := #Ctrl.Rulliera.Ax_1_2_Vel_CarroTesta AND #CIn.CarroPareggTesta.Sens.FTC_Ingombro_Ing;
   IF #_w1 AND NOT #Ctrl.Rulliera.Ax_2_MemoRall THEN
       #Ctrl.Rulliera.SP_TimeMemoRall := "Feed2Stopper_DelayVel0Calc"(Sensor_Distance_mm := 265.0,
                               Conveyor_Vel_mm_min := "A0302_Rulliera".COut.Ax_2.ActualVelocity,
                               Conveyor_Dec_mm_s2 := "A0302_Rulliera_PERS".Par.Ax_Aut.Aut_Dec);
   END_IF;
   IF #_w1 THEN #Ctrl.Rulliera.Ax_2_MemoRall := TRUE; END_IF;
   #Ctrl.Rulliera.TON_RitardoRallenta.TON(IN := #Ctrl.Rulliera.Ax_2_MemoRall,
                           PT := #Ctrl.Rulliera.SP_TimeMemoRall);
   IF #Ctrl.Rulliera.TON_RitardoRallenta.Q AND ("A0302_Rulliera".COut.Ax_2.ActualVelocity > 100.0) THEN
       #Ctrl.Rulliera.Ax_1_2_Vel_ZeroTesta := TRUE;
   END_IF;
   IF #Ctrl.Rulliera.Ax_1_2_Vel_ZeroTesta AND ("A0302_Rulliera".COut.Ax_2.ActualVelocity < 100.0) THEN
       #Ctrl.Rulliera.Ax_1_2_End_VelZero := TRUE;
   END_IF;
   IF #Ctrl.Rulliera.Ax_1_2_End_VelZero AND (NOT #CIn.CarroPareggTesta.Sens.FTC_Prox_Ls OR NOT #CIn.CarroPareggCoda.Sens.FTC_Ingombro_Out) THEN
       #Ctrl.Rulliera.Ax_1_2_Vel_Appoggio := TRUE;
   END_IF;
   IF NOT #Ctrl.Rulliera.Ax_1_2_Vel_CarroTesta THEN
       #Ctrl.Rulliera.Ax_2_MemoRall := FALSE;
       #Ctrl.Rulliera.Ax_1_2_Vel_ZeroTesta := FALSE;
       #Ctrl.Rulliera.Ax_1_2_End_VelZero := FALSE;
       #Ctrl.Rulliera.Ax_1_2_Vel_Appoggio := FALSE;
   END_IF;
END_REGION

REGION Network 43: [Ax] Rulliera - COut Manager
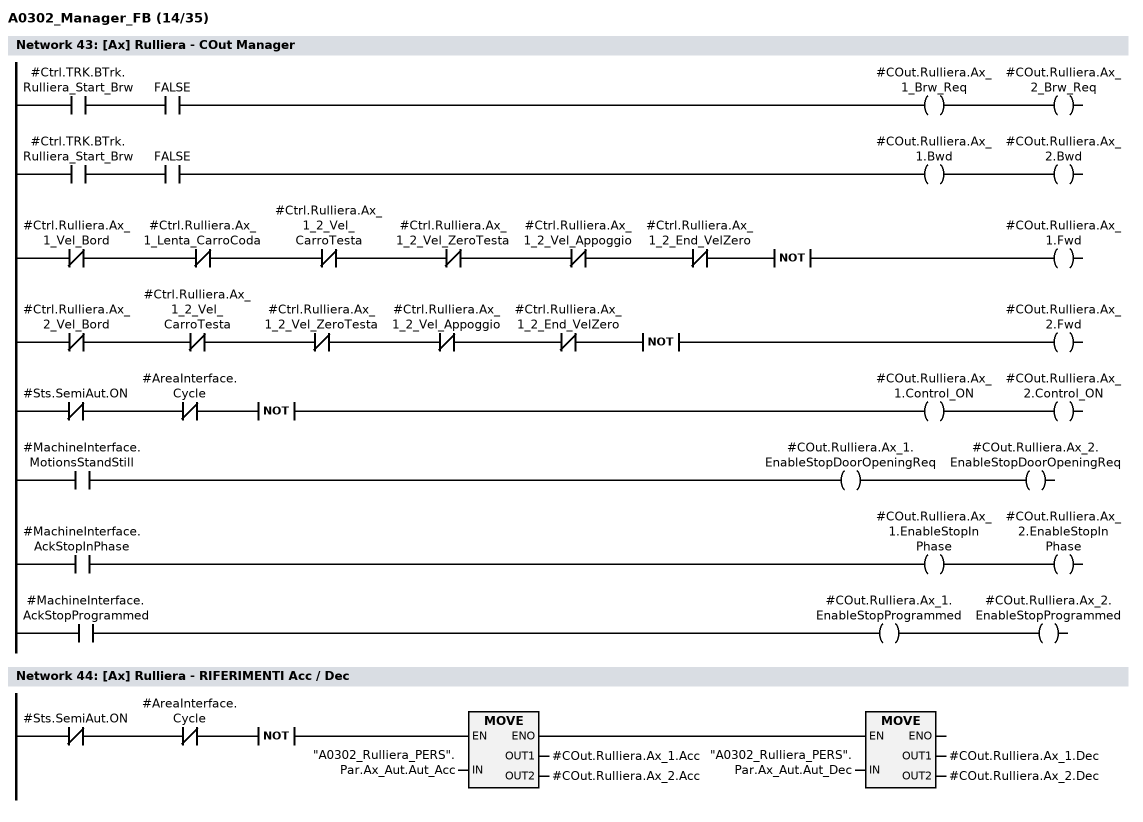
   RUNG wire#powerrail
      Contact( #Ctrl.TRK.BTrk.Rulliera_Start_Brw )
      Contact( FALSE )
      Coil( #COut.Rulliera.Ax_1_Brw_Req )
      Coil( #COut.Rulliera.Ax_2_Brw_Req )
   END_RUNG
   RUNG wire#powerrail
      Contact( #Ctrl.TRK.BTrk.Rulliera_Start_Brw )
      Contact( FALSE )
      Coil( #COut.Rulliera.Ax_1.Bwd )
      Coil( #COut.Rulliera.Ax_2.Bwd )
   END_RUNG
   RUNG wire#powerrail
      I_Contact( #Ctrl.Rulliera.Ax_1_Vel_Bord )
      I_Contact( #Ctrl.Rulliera.Ax_1_Lenta_CarroCoda )
      I_Contact( #Ctrl.Rulliera.Ax_1_2_Vel_CarroTesta )
      I_Contact( #Ctrl.Rulliera.Ax_1_2_Vel_ZeroTesta )
      I_Contact( #Ctrl.Rulliera.Ax_1_2_Vel_Appoggio )
      I_Contact( #Ctrl.Rulliera.Ax_1_2_End_VelZero )
      Not()
      Coil( #COut.Rulliera.Ax_1.Fwd )
   END_RUNG
   RUNG wire#powerrail
      I_Contact( #Ctrl.Rulliera.Ax_2_Vel_Bord )
      I_Contact( #Ctrl.Rulliera.Ax_1_2_Vel_CarroTesta )
      I_Contact( #Ctrl.Rulliera.Ax_1_2_Vel_ZeroTesta )
      I_Contact( #Ctrl.Rulliera.Ax_1_2_Vel_Appoggio )
      I_Contact( #Ctrl.Rulliera.Ax_1_2_End_VelZero )
      Not()
      Coil( #COut.Rulliera.Ax_2.Fwd )
   END_RUNG
   RUNG wire#powerrail
      I_Contact( #Sts.SemiAut.ON )
      I_Contact( #AreaInterface.Cycle )
      Not()
      Coil( #COut.Rulliera.Ax_1.Control_ON )
      Coil( #COut.Rulliera.Ax_2.Control_ON )
   END_RUNG
   RUNG wire#powerrail
      Contact( #MachineInterface.MotionsStandStill )
      Coil( #COut.Rulliera.Ax_1.EnableStopDoorOpeningReq )
      Coil( #COut.Rulliera.Ax_2.EnableStopDoorOpeningReq )
   END_RUNG
   RUNG wire#powerrail
      Contact( #MachineInterface.AckStopInPhase )
      Coil( #COut.Rulliera.Ax_1.EnableStopInPhase )
      Coil( #COut.Rulliera.Ax_2.EnableStopInPhase )
   END_RUNG
   RUNG wire#powerrail
      Contact( #MachineInterface.AckStopProgrammed )
      Coil( #COut.Rulliera.Ax_1.EnableStopProgrammed )
      Coil( #COut.Rulliera.Ax_2.EnableStopProgrammed )
   END_RUNG
   // the same network as SCL:
   #COut.Rulliera.Ax_1_Brw_Req := #Ctrl.TRK.BTrk.Rulliera_Start_Brw AND FALSE;
   #COut.Rulliera.Ax_2_Brw_Req := #COut.Rulliera.Ax_1_Brw_Req;
   #COut.Rulliera.Ax_1.Bwd := #Ctrl.TRK.BTrk.Rulliera_Start_Brw AND FALSE;
   #COut.Rulliera.Ax_2.Bwd := #COut.Rulliera.Ax_1.Bwd;
   #COut.Rulliera.Ax_1.Fwd := NOT (NOT #Ctrl.Rulliera.Ax_1_Vel_Bord AND NOT #Ctrl.Rulliera.Ax_1_Lenta_CarroCoda AND NOT #Ctrl.Rulliera.Ax_1_2_Vel_CarroTesta AND NOT #Ctrl.Rulliera.Ax_1_2_Vel_ZeroTesta AND NOT #Ctrl.Rulliera.Ax_1_2_Vel_Appoggio AND NOT #Ctrl.Rulliera.Ax_1_2_End_VelZero);
   #COut.Rulliera.Ax_2.Fwd := NOT (NOT #Ctrl.Rulliera.Ax_2_Vel_Bord AND NOT #Ctrl.Rulliera.Ax_1_2_Vel_CarroTesta AND NOT #Ctrl.Rulliera.Ax_1_2_Vel_ZeroTesta AND NOT #Ctrl.Rulliera.Ax_1_2_Vel_Appoggio AND NOT #Ctrl.Rulliera.Ax_1_2_End_VelZero);
   #COut.Rulliera.Ax_1.Control_ON := NOT (NOT #Sts.SemiAut.ON AND NOT #AreaInterface.Cycle);
   #COut.Rulliera.Ax_2.Control_ON := #COut.Rulliera.Ax_1.Control_ON;
   #COut.Rulliera.Ax_1.EnableStopDoorOpeningReq := #MachineInterface.MotionsStandStill;
   #COut.Rulliera.Ax_2.EnableStopDoorOpeningReq := #MachineInterface.MotionsStandStill;
   #COut.Rulliera.Ax_1.EnableStopInPhase := #MachineInterface.AckStopInPhase;
   #COut.Rulliera.Ax_2.EnableStopInPhase := #MachineInterface.AckStopInPhase;
   #COut.Rulliera.Ax_1.EnableStopProgrammed := #MachineInterface.AckStopProgrammed;
   #COut.Rulliera.Ax_2.EnableStopProgrammed := #MachineInterface.AckStopProgrammed;
END_REGION

REGION Network 44: [Ax] Rulliera - RIFERIMENTI Acc / Dec
   RUNG wire#powerrail
      I_Contact( #Sts.SemiAut.ON )
      I_Contact( #AreaInterface.Cycle )
      Not()
      Move(in := "A0302_Rulliera_PERS".Par.Ax_Aut.Aut_Acc, out1 => #COut.Rulliera.Ax_1.Acc, out2 => #COut.Rulliera.Ax_2.Acc)
      Move(in := "A0302_Rulliera_PERS".Par.Ax_Aut.Aut_Dec, out1 => #COut.Rulliera.Ax_1.Dec, out2 => #COut.Rulliera.Ax_2.Dec)
   END_RUNG
   // the same network as SCL:
   IF NOT (NOT #Sts.SemiAut.ON AND NOT #AreaInterface.Cycle) THEN
       #COut.Rulliera.Ax_1.Acc := "A0302_Rulliera_PERS".Par.Ax_Aut.Aut_Acc;
       #COut.Rulliera.Ax_2.Acc := "A0302_Rulliera_PERS".Par.Ax_Aut.Aut_Acc;
       #COut.Rulliera.Ax_1.Dec := "A0302_Rulliera_PERS".Par.Ax_Aut.Aut_Dec;
       #COut.Rulliera.Ax_2.Dec := "A0302_Rulliera_PERS".Par.Ax_Aut.Aut_Dec;
   END_IF;
END_REGION

REGION Network 45 (SCL): [Ax] Rulliera - RIFERIMENTI Velocità
   #COut.Rulliera.Ax_1.Vel := 0.0;
   #COut.Rulliera.Ax_2.Vel := 0.0;

   // RIFERIMENTI VELOCITà
   IF #Ctrl.Rulliera.Ax_1_2_Vel_Appoggio THEN
       #COut.Rulliera.Ax_1.Vel := #COut.Rulliera.Ax_2.Vel := 5000.0;

   ELSIF #Ctrl.Rulliera.Ax_1_2_Vel_ZeroTesta AND NOT #Ctrl.Rulliera.Ax_1_2_End_VelZero THEN
       #COut.Rulliera.Ax_1.Vel := #COut.Rulliera.Ax_2.Vel := 0.0;

   ELSIF #Ctrl.Rulliera.Ax_1_2_Vel_CarroTesta THEN
       #COut.Rulliera.Ax_1.Vel :=   #COut.Rulliera.Ax_2.Vel := "A0302_Rulliera_PERS".Par.Ax_Aut.Aut_Vel;

   ELSIF #Ctrl.Rulliera.Ax_1_Lenta_CarroCoda THEN
       #COut.Rulliera.Ax_1.Vel := 2000.0;

   ELSIF #Ctrl.Rulliera.Ax_1_Vel_Bord THEN
       #COut.Rulliera.Ax_1.Vel := "A0302_Bordatrice".COut.Ax.ActualVelocity;

       IF #Ctrl.Rulliera.Ax_2_Vel_Bord THEN
           #COut.Rulliera.Ax_2.Vel := "A0302_Bordatrice".COut.Ax.ActualVelocity;
       END_IF;
   END_IF;
END_REGION

REGION Network 47: <<< POSIZIONAMENTO CARRI >>>
END_REGION

REGION Network 48 (SCL): == Zona Pareggiatori Vuota ==
   REGION CONTROLLO CHE CI SIANO LE CONDIZIONI PER MUOVERSI IN ENTRATA A0302 (TRK EMPTY)
       // Controllo zona libera dai traking e sensori non in lettura su Spintore e Bordatrice in uscita su rulliera
       // 
       FOR #i := 1 TO "BTRK_A0302_ENTRY_ITEMS" DO
           IF "BTrk".A0302_ENTRY.B[#i].B_ID = 0 THEN
               #Sts.BTrk.A0302Entry_Absence := TRUE;
           ELSE
               #Sts.BTrk.A0302Entry_Absence := FALSE;
               EXIT;
           END_IF;
       END_FOR;

       // Verifica se BTrk assente e sensori su rulliera di coda non in lettura
       #Sts.BTrk.ZoneA0302Entry_Empty := (#Sts.BTrk.A0302Entry_Absence AND NOT #CIn.Rulliera.Coda.Sens.FTC_Rall
       AND NOT #CIn.Bordatrice.Sens.FTC_Ingresso AND NOT #CIn.Bordatrice.Sens.FTC_Uscita);

   END_REGION


   REGION CONTROLLO CHE CI SIANO LE CONDIZIONI PER MUOVERSI IN USCITA A0302 (TRK EMPTY)
       // Controllo zona libera dai traking e sensori non in lettura su rulliera per movimento Carri Pareggiatori
       // 
       FOR #i := 1 TO "BTRK_A0302_EXIT_ITEMS" DO
           IF "BTrk".A0302_EXIT.B[#i].B_ID = 0 THEN
               #Sts.BTrk.A0302Exit_Absence := TRUE;
           ELSE
               #Sts.BTrk.A0302Exit_Absence := FALSE;
               EXIT;
           END_IF;
       END_FOR;

       // Verifica se BTrk assente e sensori su rulliera di centro + dei carri pareggiatori di testa e coda non in lettura
       #Sts.BTrk.ZoneA0302Exit_Empty := (#Sts.BTrk.A0302Exit_Absence
       AND NOT #CIn.Rulliera.Centro.Sens.FTC_Centrale                                                                   // Sensori rulliera avanzamento Beams
       AND NOT #CIn.CarroPareggCoda.Sens.PresenzaMat AND NOT #CIn.CarroPareggTesta.Sens.PresenzaMat                     // Sensori presenza Beams su manipolatori
       AND NOT #CIn.CarroPareggTesta.Sens.FTC_Ingombro_Ing AND NOT #CIn.CarroPareggTesta.Sens.FTC_Prox_Ls               // Sensori presenza Beams su carro di testa
       AND NOT #CIn.CarroPareggCoda.Sens.FTC_Ingombro_Ing AND NOT #CIn.CarroPareggCoda.Sens.FTC_Ingombro_Out);          // Sensori presenza Beams su carro di coda

   END_REGION
END_REGION

REGION Network 49 (SCL): == Calcolo setpoint posizione carri in funzione della cremaliera ==
   // Foglio di calcolo posizione Cremaliera fornito
   // 

   #CarroTesta.PosBattutePz := 348.56;



   IF "BTrk".A0302_EXIT.Beam_Len > 0 THEN
       // *****  Calcolo CARRO di TESTA ******
       #CarroTesta.SemiBeamLen := ("BTrk".A0302_EXIT.Beam_Len / 2.0);
       #CarroTesta.PosBattutePz := #Par.CarroPareggTesta.Preset;
       #CarroTesta.RimanenzaPos := (#CarroTesta.SemiBeamLen - #CarroTesta.PosBattutePz);
       #CarroTesta.NrPassiReq := (#CarroTesta.RimanenzaPos / #Par.Cremaliera.Passo);

       // Calcolo i numeri di passi cremaliera richiesti per spostarmi della rimanenza
       #CarroTesta.PassoReq := ROUND(#CarroTesta.NrPassiReq);

       // ***** Calcolo CARRO di CODA *****
       #CarroCoda.SemiBeamLen := ("BTrk".A0302_EXIT.Beam_Len / 2.0);
       #CarroCoda.PosBattutePz := (#Par.CarroPareggCoda.Preset - "A0302_PareggiatoreCoda_PERS".Par_Sens.AI.RangeLow);
       #CarroCoda.RimanenzaPos := ("BTrk".A0302_EXIT.Beam_Len - #Ctrl.CarroPareggTesta.Ax.Pos - #CarroCoda.PosBattutePz) + ("A0302_PareggiatoreCoda_PERS".Par_Sens.AI.RangeLow +2.0);
       #CarroCoda.NrPassiReq := (#CarroCoda.RimanenzaPos / #Par.Cremaliera.Passo);

       // Calcolo i numeri di passi cremaliera richiesti per spostarmi della rimanenza
       #CarroCoda.PassoReq := ROUND(#CarroCoda.NrPassiReq);

       // Calcolo del setpoint di posizione dei 2 carri in funzione della misura calcolata - Se cambia il Beam Len viene richiesto il nuovo riposizionamento
       #Ctrl.CarroPareggTesta.Ax.Pos := (#CarroTesta.PassoReq * #Par.Cremaliera.Passo) + #CarroTesta.PosBattutePz;
       #Ctrl.CarroPareggCoda.Ax.Pos := (#CarroCoda.PassoReq * #Par.Cremaliera.Passo) + #CarroCoda.PosBattutePz + "A0302_PareggiatoreCoda_PERS".Par_Sens.AI.RangeLow;
   END_IF;
END_REGION

REGION Network 50 (SCL): == Controllo posizionamento dei carri rispetto alle spalle ==
   //

   REGION ********* Carro di TESTA ***********
       //Controllo che ci sia sempre la distanza minima tra il pareggiatore e la spalla di Testa quando muovo in direzione FRW(Apertura)
       //
       IF NOT #CIn.CarroPareggTesta.Ax_InWPos AND NOT #Sts.Attrezzamento.Ready THEN

           #Ctrl.CarroPareggTesta.Ax.MoveToPos := #Sts.Attrezzamento.RequestNewPosition AND #Sts.BTrk.ZoneA0302Exit_Empty;

       ELSIF #Sts.Attrezzamento.Ready THEN

           #Ctrl.CarroPareggTesta.Ax.MoveToPos := FALSE;
       END_IF;
   END_REGION


   REGION ********* Carro di CODA ***********
       //Controllo che ci sia sempre la distanza minima tra il pareggiatore e la spalla di Coda quando muovo in direzione FRW(Apertura)
       IF NOT #CIn.CarroPareggCoda.Ax_InWPos AND NOT #Sts.Attrezzamento.Ready THEN

           #Ctrl.CarroPareggCoda.Ax.MoveToPos := #Sts.Attrezzamento.RequestNewPosition AND #Sts.BTrk.ZoneA0302Exit_Empty;

       ELSIF #Sts.Attrezzamento.Ready THEN

           #Ctrl.CarroPareggCoda.Ax.MoveToPos := FALSE;
       END_IF;
   END_REGION

   // Controllo Attrezzaggio pronto 
   // Se sono con tutti e 2 i carri in finestra resetto la richiesta di nuova posizione
   IF #CIn.CarroPareggCoda.Ax_InWPos AND #CIn.CarroPareggTesta.Ax_InWPos  AND #CIn.CarroPareggCoda.Bloccaggio.Work AND #CIn.CarroPareggTesta.Bloccaggio.Work THEN
       #Sts.Attrezzamento.Ready := TRUE;
   ELSE
       #Sts.Attrezzamento.Ready := FALSE;
   END_IF;
END_REGION

REGION Network 51: ************************************************************************************
END_REGION

REGION Network 53: *************************************************************************************
END_REGION

REGION Network 54: <<<< PAREGGIATORE TESTA >>>>
END_REGION

REGION Network 55: <+>
END_REGION

